(* IEC 61131-3 sources: SmartHomeNew/snapshots/2026-05-19 (part 5) *)

(* ---- PRG_Heating.st ---- *)
PROGRAM PRG_Heating
VAR
    fbHeatingManager : FB_Heating_System_Manager;
    fbDHWManager : FB_DHW_Manager;
    fbDiagnosticsPhase : FB_Heating_Runtime_Diagnostics_Phase;
    fbObserverPhase : FB_Heating_Runtime_Observer_Phase;
    fbMetaSupervisionPublisher : FB_Heating_Runtime_Meta_Supervision_Publisher;
    fbExplainabilityPublisher : FB_Heating_Runtime_Explainability_Publisher;
    fbServiceGatingPhase : FB_Heating_Runtime_Service_Gating_Phase;
    fbStatePublicationPhase : FB_Heating_Runtime_State_Publication_Phase;
    fbOutputProjectionPhase : FB_Heating_Runtime_Output_Projection_Phase;

    L_Runtime_Context : ST_Heating_Runtime_Context;

    L_i : INT;
    L_Current_Hour : UINT;
    L_Boiler_Modulation_REAL : ARRAY[1..GVL_CONSTANTS.C_MAX_BOILERS] OF REAL;
    L_Room_Temps_Normalized : ARRAY[1..GVL_CONSTANTS.C_MAX_ZONES] OF REAL;
    L_Floor_Temps_Normalized : ARRAY[1..GVL_CONSTANTS.C_MAX_HEATING_CIRCUITS] OF REAL;
    L_Outdoor_Temp_Normalized : REAL;

    L_Heating_Emergency_Stop : BOOL;
    L_Heating_Gas_Safety_Stop : BOOL;

    L_Distributed_Execute_Allowed : BOOL;
    L_Distributed_Orchestrate_Allowed : BOOL;
    L_Distributed_Projection_Allowed : BOOL;

    L_Zone_Valves : ARRAY[1..GVL_CONSTANTS.C_MAX_HEATING_CIRCUITS] OF BOOL;
    L_Manifold_Pumps : ARRAY[1..GVL_CONSTANTS.C_MAX_MANIFOLDS] OF BOOL;
    L_Manifold_Valves : ARRAY[1..GVL_CONSTANTS.C_MAX_MANIFOLDS] OF REAL;
    L_Boiler_OT_Enable : ARRAY[1..GVL_CONSTANTS.C_MAX_BOILERS] OF BOOL;
    L_Boiler_OT_Setpoint : ARRAY[1..GVL_CONSTANTS.C_MAX_BOILERS] OF REAL;
    L_Backup_Circulation_Pump : BOOL;
    L_Electric_Heater_Enable : BOOL;
    L_Freeze_Risk_Status : BOOL;
    L_Manifold_Status : ARRAY[1..GVL_CONSTANTS.C_MAX_MANIFOLDS] OF ST_Manifold_Status;
    L_Boiler_Status : ARRAY[1..GVL_CONSTANTS.C_MAX_BOILERS] OF ST_Boiler_Status;
    L_DHW_Heating_Pump : BOOL;
    L_DHW_Circ_Pump : BOOL;
    L_DHW_Status : ST_DHW_Status;
END_VAR

FOR L_i := 1 TO GVL_CONSTANTS.C_MAX_BOILERS DO
    L_Boiler_Modulation_REAL[L_i] := TO_REAL(GVL_IO.AI_Boiler_Modulation[L_i]);
END_FOR;

L_Current_Hour := TO_UINT(GVL_TIME_SERVICE.G_Time_Of_Day_MS / 3600000);

L_Outdoor_Temp_Normalized := GVL_INPUT.IN_Outdoor_Temp;

FOR L_i := 1 TO GVL_CONSTANTS.C_MAX_ZONES DO
    L_Room_Temps_Normalized[L_i] := GVL_INPUT.IN_Room_Temps[L_i];
END_FOR;

FOR L_i := 1 TO GVL_CONSTANTS.C_MAX_HEATING_CIRCUITS DO
    L_Floor_Temps_Normalized[L_i] := GVL_INPUT.IN_Floor_Temps[L_i];
END_FOR;

L_Heating_Emergency_Stop := GVL_COMMAND_SHADOW.G_Heating_Emergency_Stop;
L_Heating_Gas_Safety_Stop := GVL_COMMAND_SHADOW.G_Heating_Gas_Safety_Stop OR GVL_STATE.G_Safety_Gas_Latched;

// Centralized distributed runtime governance.
// Freeze protection and gas safety semantics remain authoritative.
L_Distributed_Execute_Allowed :=
    GVL_Distributed_Execution_Gates.G_Can_Execute;

L_Distributed_Orchestrate_Allowed :=
    GVL_Distributed_Execution_Gates.G_Can_Orchestrate;

L_Distributed_Projection_Allowed :=
    GVL_Distributed_Execution_Gates.G_Can_Own_Projection;

L_Runtime_Context.Runtime_Enabled := TRUE;
L_Runtime_Context.Runtime_Ready := TRUE;
L_Runtime_Context.Runtime_Fault := FALSE;
L_Runtime_Context.Current_Phase := E_Heating_Runtime_Phase.HRP_IDLE;

L_Runtime_Context.Allow_DHW_Phase :=
    L_Distributed_Execute_Allowed;

L_Runtime_Context.Allow_Heating_Phase :=
    L_Distributed_Orchestrate_Allowed;

L_Runtime_Context.Allow_Service_Gating_Phase := TRUE;
L_Runtime_Context.Allow_State_Publication_Phase := TRUE;
L_Runtime_Context.Allow_Diagnostics_Phase := TRUE;

L_Runtime_Context.Allow_Output_Projection_Phase :=
    L_Distributed_Projection_Allowed;

L_Runtime_Context.DHW_Executed := FALSE;
L_Runtime_Context.Heating_Executed := FALSE;
L_Runtime_Context.Service_Gating_Executed := FALSE;
L_Runtime_Context.State_Publication_Executed := FALSE;
L_Runtime_Context.Diagnostics_Executed := FALSE;
L_Runtime_Context.Output_Projection_Executed := FALSE;

L_Runtime_Context.DHW_Before_Heating_Valid := TRUE;
L_Runtime_Context.State_Publication_Before_Diagnostics_Valid := TRUE;
L_Runtime_Context.Output_Projection_Last_Valid := TRUE;

L_Runtime_Context.Diagnostics_Isolation_Valid := TRUE;
L_Runtime_Context.Explainability_Isolation_Valid := TRUE;
L_Runtime_Context.Safety_Isolation_Valid := TRUE;
L_Runtime_Context.OpenTherm_Ownership_Valid := TRUE;
L_Runtime_Context.Cascade_Ownership_Valid := TRUE;

IF NOT L_Distributed_Execute_Allowed THEN
    L_Runtime_Context.Runtime_Status_Code := 20;
    L_Runtime_Context.Runtime_Status_Text :=
        'Heating runtime blocked by distributed governance';
ELSE
    L_Runtime_Context.Runtime_Status_Code := 1;
    L_Runtime_Context.Runtime_Status_Text :=
        'Heating runtime nominal';
END_IF;

L_Runtime_Context.Current_Phase := E_Heating_Runtime_Phase.HRP_IDLE;

fbObserverPhase(
    VI_Authorization_Stage := TRUE,
    VI_Finalization_Stage := FALSE,
    VI_Runtime_Context := L_Runtime_Context,
    VI_Diagnostics_Valid := TRUE
);

IF L_Distributed_Execute_Allowed THEN

    L_Runtime_Context.Current_Phase := E_Heating_Runtime_Phase.HRP_DHW;

    fbDHWManager(
        VI_System_Time_MS := GVL_STATUS.G_System_Time_MS,
        VI_Current_TOD := GVL_STATUS.G_Current_TOD,
        VI_IsActivePLC := GVL_STATUS.G_Is_Active_PLC,
        VI_Temp := GVL_STATE.G_DHW_Temp,
        VI_Pressure := GVL_STATE.G_DHW_Pressure,
        VI_Config := GVL_CONFIG.G_DHW_Config,
        VI_Current_Day_Of_Week := GVL_STATUS.G_Current_Day,
        VI_IO_Modules_Online := GVL_STATUS.G_IO_Modules_Online,
        VI_Reset_Errors := GVL_INTENT_USER.I_Reset_Errors,
        VI_Emergency_Stop := L_Heating_Emergency_Stop,
        VI_System_Mode := GVL_STATE.G_System_Mode,
        VO_Status => L_DHW_Status,
        VO_Heating_Pump => L_DHW_Heating_Pump,
        VO_Circ_Pump => L_DHW_Circ_Pump
    );

    L_Runtime_Context.DHW_Executed := TRUE;

END_IF;

IF L_Heating_Gas_Safety_Stop THEN
    L_DHW_Heating_Pump := FALSE;
    L_DHW_Status.Heating_Pump_On := FALSE;
END_IF;

IF L_Distributed_Orchestrate_Allowed THEN

    L_Runtime_Context.Current_Phase := E_Heating_Runtime_Phase.HRP_HEATING;

    fbHeatingManager(
        VI_System_Mode := GVL_STATE.G_System_Mode,
        VI_System_Time_MS := GVL_STATUS.G_System_Time_MS,
        VI_IsActivePLC := GVL_STATUS.G_Is_Active_PLC,
        VI_Outdoor_Temp := L_Outdoor_Temp_Normalized,
        VI_Config := GVL_CONFIG.G_Heating_Config,
        VI_Tariff := GVL_CONFIG.G_HMI_Tariff_Settings,
        VI_Current_Hour := L_Current_Hour,
        VI_DHW_Heating_Demand := L_DHW_Heating_Pump,
        VI_DHW_Target_Temp := GVL_CONFIG.G_DHW_Config.Target_Temp,
        VI_Emergency_Stop := L_Heating_Emergency_Stop,
        VI_Gas_Safety_Stop := L_Heating_Gas_Safety_Stop,
        VI_Boiler_Error_Status := GVL_STATE.G_Boiler_Error,
        VI_Boiler_OT_Online := GVL_STATE.G_Boiler_OT_Online,
        VI_Boiler_Modulation := L_Boiler_Modulation_REAL,
        VI_Floor_Temps := L_Floor_Temps_Normalized,
        VI_Room_Temps := L_Room_Temps_Normalized,
        VI_Manifold_Pressures := GVL_STATE.G_Manifold_Pressures,
        VI_Manifold_Currents := GVL_STATE.G_Manifold_Currents,
        VI_Manifold_Temps_Supply := GVL_STATE.G_Manifold_T_Supply,
        VI_Manifold_Temps_Return := GVL_STATE.G_Manifold_T_Return,
        VI_Boiler_Flame_Status := GVL_STATE.G_Boiler_Flame,
        VI_Zone_Configs := GVL_CONFIG.G_HMI_FloorHeating_Configs,
        VI_Rule_Actions := GVL_STATE.G_Rule_Actions,
        VI_IO_Modules_Online := GVL_STATUS.G_IO_Modules_Online,
        VI_Manifold_End_Switches := GVL_STATE.G_Manifold_End_Switches,
        VI_Valve_Test_Config := GVL_CONFIG.G_Valve_Test_Config,
        VO_Manifold_Valves => L_Manifold_Valves,
        VO_Manifold_Pumps => L_Manifold_Pumps,
        VO_Zone_Valves => L_Zone_Valves,
        VO_Boiler_OT_Enable => L_Boiler_OT_Enable,
        VO_Boiler_OT_Setpoint => L_Boiler_OT_Setpoint,
        VO_Backup_Circulation_Pump => L_Backup_Circulation_Pump,
        VO_Electric_Heater_Enable => L_Electric_Heater_Enable,
        VO_Freeze_Risk_Status => L_Freeze_Risk_Status,
        VO_Status => L_Manifold_Status,
        VO_Boiler_Status => L_Boiler_Status
    );

    L_Runtime_Context.Heating_Executed := TRUE;

END_IF;

L_Runtime_Context.Current_Phase := E_Heating_Runtime_Phase.HRP_SERVICE_GATING;

fbServiceGatingPhase(
    VI_Enable := TRUE,
    VIO_Manifold_Pumps := L_Manifold_Pumps,
    VIO_Backup_Circulation_Pump := L_Backup_Circulation_Pump,
    VIO_Electric_Heater_Enable := L_Electric_Heater_Enable,
    VIO_DHW_Heating_Pump := L_DHW_Heating_Pump,
    VIO_DHW_Circ_Pump := L_DHW_Circ_Pump,
    VIO_DHW_Status := L_DHW_Status,
    VIO_Freeze_Risk_Status := L_Freeze_Risk_Status
);

L_Runtime_Context.Service_Gating_Executed := fbServiceGatingPhase.VO_Executed;
L_Runtime_Context.Safety_Isolation_Valid := fbServiceGatingPhase.VO_Valid;

L_Runtime_Context.Current_Phase := E_Heating_Runtime_Phase.HRP_STATE_PUBLICATION;

fbStatePublicationPhase(
    VI_Enable := TRUE,
    VI_Zone_Valves := L_Zone_Valves,
    VI_Manifold_Pumps := L_Manifold_Pumps,
    VI_Manifold_Valves := L_Manifold_Valves,
    VI_Boiler_OT_Enable := L_Boiler_OT_Enable,
    VI_Boiler_OT_Setpoint := L_Boiler_OT_Setpoint,
    VI_Backup_Circulation_Pump := L_Backup_Circulation_Pump,
    VI_Electric_Heater_Enable := L_Electric_Heater_Enable,
    VI_Freeze_Risk_Status := L_Freeze_Risk_Status,
    VI_Manifold_Status := L_Manifold_Status,
    VI_Boiler_Status := L_Boiler_Status,
    VI_DHW_Heating_Pump := L_DHW_Heating_Pump,
    VI_DHW_Circ_Pump := L_DHW_Circ_Pump,
    VI_DHW_Status := L_DHW_Status
);

L_Runtime_Context.State_Publication_Executed := fbStatePublicationPhase.VO_Executed;
L_Runtime_Context.State_Publication_Before_Diagnostics_Valid := fbStatePublicationPhase.VO_Valid;

L_Runtime_Context.Current_Phase := E_Heating_Runtime_Phase.HRP_DIAGNOSTICS;

fbDiagnosticsPhase(
    VI_Enable := TRUE,
    VI_System_Time_MS := GVL_STATUS.G_System_Time_MS
);

L_Runtime_Context.Diagnostics_Executed := fbDiagnosticsPhase.VO_Executed;
L_Runtime_Context.Diagnostics_Isolation_Valid := fbDiagnosticsPhase.VO_Valid;

fbObserverPhase(
    VI_Authorization_Stage := FALSE,
    VI_Finalization_Stage := TRUE,
    VI_Runtime_Context := L_Runtime_Context,
    VI_Diagnostics_Valid := L_Runtime_Context.Diagnostics_Isolation_Valid
);

fbMetaSupervisionPublisher(
    VI_Enable := TRUE,
    VI_Runtime_Observation_Valid := GVL_Heating_Runtime_Observation.G_Runtime_Observation_Valid,
    VI_Runtime_Observer_Ready := GVL_Heating_Runtime_Observation.G_Runtime_Observer_Ready,
    VI_Runtime_Observer_Fault := GVL_Heating_Runtime_Observation.G_Runtime_Observer_Fault,
    VI_Runtime_Status_Code := GVL_Heating_Runtime_Observation.G_Runtime_Observation_Status_Code,
    VI_Runtime_Status_Text := GVL_Heating_Runtime_Observation.G_Runtime_Observation_Status_Text
);

GVL_Heating_Runtime_Meta.G_Runtime_Meta_Supervision :=
    fbMetaSupervisionPublisher.VO_Meta;

GVL_Heating_Runtime_Meta.G_Runtime_Meta_Publication_Valid :=
    fbMetaSupervisionPublisher.VO_Publication_Valid;

GVL_Heating_Runtime_Meta.G_Runtime_Meta_Status_Code :=
    fbMetaSupervisionPublisher.VO_Meta.Status_Code;

GVL_Heating_Runtime_Meta.G_Runtime_Meta_Status_Text :=
    fbMetaSupervisionPublisher.VO_Meta.Status_Text;

fbExplainabilityPublisher(
    VI_Enable := TRUE,
    VI_System_Time_MS := GVL_STATUS.G_System_Time_MS,
    VI_Runtime_Context := L_Runtime_Context,
    VI_Runtime_Observation_Valid := GVL_Heating_Runtime_Observation.G_Runtime_Observation_Valid,
    VI_Runtime_Observer_Fault := GVL_Heating_Runtime_Observation.G_Runtime_Observer_Fault,
    VI_Runtime_Status_Code := GVL_Heating_Runtime_Observation.G_Runtime_Observation_Status_Code,
    VI_Runtime_Status_Text := GVL_Heating_Runtime_Observation.G_Runtime_Observation_Status_Text
);

GVL_Heating_Runtime_Explainability.G_Runtime_Phase_Event :=
    fbExplainabilityPublisher.VO_Phase_Event;

GVL_Heating_Runtime_Explainability.G_Runtime_Anomaly :=
    fbExplainabilityPublisher.VO_Anomaly;

GVL_Heating_Runtime_Explainability.G_Runtime_Blackbox_Event :=
    fbExplainabilityPublisher.VO_Blackbox_Event;

GVL_Heating_Runtime_Explainability.G_Runtime_Blackbox_Timeline :=
    fbExplainabilityPublisher.VO_Blackbox_Timeline;

GVL_Heating_Runtime_Explainability.G_Runtime_Event_Buffer :=
    fbExplainabilityPublisher.VO_Event_Buffer;

GVL_Heating_Runtime_Explainability.G_Runtime_Adaptive_Intelligence :=
    fbExplainabilityPublisher.VO_Adaptive_Intelligence;

GVL_Heating_Runtime_Explainability.G_Runtime_Causality_Graph :=
    fbExplainabilityPublisher.VO_Causality_Graph;

GVL_Heating_Runtime_Explainability.G_Runtime_Explainability_Publication_Valid :=
    fbExplainabilityPublisher.VO_Publication_Valid;

GVL_Heating_Runtime_Explainability.G_Runtime_Explainability_Status_Code :=
    fbExplainabilityPublisher.VO_Phase_Event.Status_Code;

GVL_Heating_Runtime_Explainability.G_Runtime_Explainability_Status_Text :=
    fbExplainabilityPublisher.VO_Phase_Event.Status_Text;

IF L_Distributed_Projection_Allowed THEN

    L_Runtime_Context.Current_Phase := E_Heating_Runtime_Phase.HRP_OUTPUT_PROJECTION;

    fbOutputProjectionPhase(
        VI_Enable := TRUE,
        VI_Zone_Valves := L_Zone_Valves,
        VI_Manifold_Pumps := L_Manifold_Pumps,
        VI_Manifold_Valves := L_Manifold_Valves,
        VI_DHW_Heating_Pump := L_DHW_Heating_Pump,
        VI_DHW_Circ_Pump := L_DHW_Circ_Pump,
        VI_Backup_Circulation_Pump := L_Backup_Circulation_Pump,
        VI_Electric_Heater_Enable := L_Electric_Heater_Enable
    );

    L_Runtime_Context.Output_Projection_Executed :=
        fbOutputProjectionPhase.VO_Executed;

    L_Runtime_Context.Output_Projection_Last_Valid :=
        fbOutputProjectionPhase.VO_Valid;

END_IF;

L_Runtime_Context.Current_Phase := E_Heating_Runtime_Phase.HRP_COMPLETE;

// >>> BULK_SYNC_ANCHOR: PRG_Heating <<<
END_PROGRAM

(* ---- PRG_Heating_Policy_Manager.st ---- *)
PROGRAM PRG_Heating_Policy_Manager
VAR
    fbPolicyManager : FB_Heating_Policy_Manager;
    fbSchedule : FB_Heating_Schedule_Preheat;
    fbThermal : FB_Heating_Thermal_Model;
    fbPredictive : FB_Heating_Predictive_Controller;
    fbOptimizer : FB_Heating_Optimizer;
    fbTime : FB_Time_Service;
    L_i : INT;
    L_Room_Avg : REAL;
    L_Floor_Avg : REAL;
END_VAR

fbTime();
fbThermal();
fbPredictive();
fbOptimizer();

L_Room_Avg := 0.0;
L_Floor_Avg := 0.0;

FOR L_i := 1 TO GVL_CONSTANTS.C_MAX_ZONES DO
    L_Room_Avg := L_Room_Avg + GVL_STATE.G_Room_Temps[L_i];
    L_Floor_Avg := L_Floor_Avg + GVL_STATE.G_Floor_Temps[L_i];
END_FOR;

L_Room_Avg := L_Room_Avg / TO_REAL(GVL_CONSTANTS.C_MAX_ZONES);
L_Floor_Avg := L_Floor_Avg / TO_REAL(GVL_CONSTANTS.C_MAX_ZONES);

fbPolicyManager(
    VI_System_Time_MS := GVL_TIME_SERVICE.G_Now_MS,
    VI_System_Mode := GVL_STATE.G_System_Mode,
    VI_RootCause := GVL_STATE.G_Heating_RootCause,
    VI_RootConfidence := GVL_STATE.G_Heating_RootConfidence,
    VI_Min_Hold_MS := GVL_CONFIG.G_Policy_Min_Hold_MS,
    VI_Emergency_Stop := GVL_STATE.G_Safety_Emergency_Stop,
    VI_Gas_Safety := GVL_STATE.G_Safety_Gas_Latched,
    VI_Room_Temp_Avg := L_Room_Avg,
    VI_Floor_Temp_Avg := L_Floor_Avg,
    VI_Supply_Temp := GVL_STATE.G_Manifold_T_Supply[1],
    VI_Return_Temp := GVL_STATE.G_Manifold_T_Return[1],
    VI_Target_Temp := GVL_STATE.G_Target_Temperature,
    VI_Room_Temps := GVL_STATE.G_Room_Temps,
    VI_Floor_Temps := GVL_STATE.G_Floor_Temps
);

fbSchedule(
    VI_System_Time_MS := GVL_TIME_SERVICE.G_Now_MS,
    VI_Time_Of_Day_MS := GVL_TIME_SERVICE.G_Time_Of_Day_MS,
    VI_Day_Of_Week := GVL_TIME_SERVICE.G_Day_Of_Week,
    VI_Enable := TRUE
);

GVL_HEATING_POLICY.G_Policy_Mode := fbPolicyManager.VO_Policy_Mode;
GVL_HEATING_POLICY.G_Policy_Block_Heating_Request := fbPolicyManager.VO_Block_Heating;
GVL_HEATING_POLICY.G_Policy_Target_Adjustment := fbPolicyManager.VO_Target_Adjustment;
GVL_HEATING_POLICY.G_Policy_Priority_Multiplier := fbPolicyManager.VO_Priority_Multiplier;
GVL_HEATING_POLICY.G_Policy_Self_Tune_Active := fbPolicyManager.VO_Self_Tune_Active;
GVL_HEATING_POLICY.G_Policy_Self_Tune_Level := fbPolicyManager.VO_Self_Tune_Level;
GVL_HEATING_POLICY.G_Policy_Feedback_Stable := fbPolicyManager.VO_Feedback_Stable;
GVL_HEATING_POLICY.G_Policy_Feedback_Improving := fbPolicyManager.VO_Feedback_Improving;
GVL_HEATING_POLICY.G_Policy_Feedback_Quality := fbPolicyManager.VO_Feedback_Quality;

END_PROGRAM

(* ---- PRG_Historical_Ordering_Integrity_Governor.st ---- *)
PROGRAM PRG_Historical_Ordering_Integrity_Governor
IF GVL_DISTRIBUTED_EPOCH_LINEARITY_FABRIC.Distributed_Epoch_Linearity_Granted
AND NOT GVL_HISTORICAL_ORDERING_INTEGRITY_FABRIC.Historical_Order_Divergence
AND NOT GVL_HISTORICAL_ORDERING_INTEGRITY_FABRIC.Unsafe_Historical_Rewrite_Detected
AND NOT GVL_HISTORICAL_ORDERING_INTEGRITY_FABRIC.Historical_Causality_Gap_Detected THEN

    GVL_HISTORICAL_ORDERING_INTEGRITY_FABRIC.Historical_Ordering_Integrity_Valid := TRUE;
    GVL_HISTORICAL_ORDERING_INTEGRITY_FABRIC.Historical_Ordering_Integrity_Granted := TRUE;
    GVL_HISTORICAL_ORDERING_INTEGRITY_FABRIC.Historical_Ordering_Integrity_Granted_Proof := TRUE;
    GVL_HISTORICAL_ORDERING_INTEGRITY_FABRIC.Historical_Timeline_Canonical := TRUE;
    GVL_HISTORICAL_ORDERING_INTEGRITY_FABRIC.Forensic_Ordering_Coherent := TRUE;
END_IF;
END_PROGRAM

(* ---- PRG_IO_Write.st ---- *)
PROGRAM PRG_IO_Write
VAR
    L_i : INT;
    L_Heating_Forced_Off : BOOL;
    L_Vent_Forced_Off : BOOL;
    L_Water_Forced_Off : BOOL;
    L_Access_Forced_Off : BOOL;
    L_Access_Safety_Override : BOOL;
    L_Global_Hard_Stop : BOOL;
    L_Gas_Safety_Stop : BOOL;
    L_Freeze_Active : BOOL;
    L_Gas_Fire_Siren_Enable : BOOL;
    L_PreOutput_Block_IO : BOOL;
    L_Output_Freshness_Block : BOOL;
    L_Output_Publication_Block : BOOL;
    L_Distributed_Publication_Block : BOOL;
    L_Snapshot_Block : BOOL;
    L_Distributed_Execution_Block : BOOL;
    L_Gas_Siren_Authority : BOOL;
    L_Fire_Siren_Authority : BOOL;
    fbTrace : FB_Trace_Write;
END_VAR

L_PreOutput_Block_IO := GVL_COMMAND_VERIFY.PreOutput_Block_IO;
L_Output_Freshness_Block := GVL_OUTPUT_EPOCH.Output_Forced_Safe_Decay;

L_Output_Publication_Block :=
    (NOT GVL_OUTPUT_EPOCH.Output_Publication_Valid)
    OR (NOT GVL_OUTPUT_EPOCH.Output_Runtime_Epoch_Valid)
    OR GVL_OUTPUT_EPOCH.Output_Lease_Expired;

// Final distributed publication continuity authority.
L_Distributed_Publication_Block :=
    (NOT GVL_DISTRIBUTED_COMMIT.Distributed_Commit_Valid)
    OR GVL_DISTRIBUTED_COMMIT.Distributed_Commit_Quarantine_Active
    OR GVL_DISTRIBUTED_COMMIT.Commit_Lease_Expired
    OR (NOT GVL_DISTRIBUTED_SNAPSHOT.Distributed_Publication_Reconciled)
    OR (NOT GVL_DISTRIBUTED_SNAPSHOT.Distributed_Publication_Freeze_Valid)
    OR (NOT GVL_DISTRIBUTED_SNAPSHOT.Distributed_Snapshot_Consistent);

L_Snapshot_Block :=
    (NOT GVL_RUNTIME_SNAPSHOT.Snapshot_Frozen)
    OR (NOT GVL_RUNTIME_SNAPSHOT.Snapshot_Publication_Allowed)
    OR (NOT GVL_RUNTIME_SNAPSHOT.Snapshot_Copy_Valid)
    OR (NOT GVL_RUNTIME_SNAPSHOT.Snapshot_Isolation_Valid)
    OR GVL_RUNTIME_SNAPSHOT.Snapshot_Mutation_Detected;

L_Distributed_Execution_Block :=
    NOT GVL_Distributed_Execution_Gates.G_Can_Execute
    OR NOT GVL_Distributed_Execution_Gates.G_Can_Own_Projection;

L_Global_Hard_Stop :=
    GVL_COMMAND_SHADOW.G_Heating_Emergency_Stop
    OR L_PreOutput_Block_IO
    OR L_Output_Freshness_Block
    OR L_Output_Publication_Block
    OR L_Distributed_Publication_Block
    OR L_Snapshot_Block
    OR L_Distributed_Execution_Block;

L_Gas_Safety_Stop := GVL_COMMAND_SHADOW.G_Heating_Gas_Safety_Stop OR GVL_COMMAND_SHADOW.G_Boiler_Stop;
L_Freeze_Active := GVL_STATE.G_Safety_Freeze_Risk;
L_Gas_Fire_Siren_Enable := GVL_ALARM.G_Gas_Fire_Siren OR GVL_ALARM.G_Global_Siren OR GVL_ALARM.G_Global_Critical;

L_Gas_Siren_Authority := GVL_HEALTH_BRIDGE.G_Gas_Detected OR GVL_HEALTH_BRIDGE.G_CO_Alarm_Level OR GVL_STATE.G_Safety_Gas_Latched;
L_Fire_Siren_Authority := GVL_HEALTH_BRIDGE.G_Smoke_Detected OR GVL_STATE.G_Safety_Smoke_Latched;

IF NOT GVL_STATUS.G_Is_Active_PLC OR L_Global_Hard_Stop THEN

    FOR L_i := 1 TO GVL_CONSTANTS.C_MAX_HEATING_CIRCUITS DO
        GVL_IO.DO_Zone_Valves[L_i] := FALSE;
    END_FOR;

    GVL_IO.DO_Gas_Valve_Close := TRUE;

    IF L_Distributed_Publication_Block THEN
        fbTrace(
            iLayer := TRACE_IO,
            iSource := SRC_IO,
            iReason := REASON_SAFETY_BLOCK,
            iValueBool := TRUE,
            iValueReal := UDINT_TO_REAL(GVL_DISTRIBUTED_COMMIT.Distributed_Commit_Last_Error_Code),
            iText := 'IO blocked by distributed publication continuity authority');
    END_IF;

    IF L_Output_Publication_Block THEN
        fbTrace(
            iLayer := TRACE_IO,
            iSource := SRC_IO,
            iReason := REASON_SAFETY_BLOCK,
            iValueBool := TRUE,
            iValueReal := UDINT_TO_REAL(GVL_OUTPUT_EPOCH.Output_Last_Error_Code),
            iText := 'IO blocked by finalized output publication authority');
    END_IF;

    RETURN;
END_IF;

fbTrace(
    iLayer := TRACE_IO,
    iSource := SRC_IO,
    iReason := REASON_DOMAIN_PROJECTION,
    iValueBool := TRUE,
    iValueReal := 0.0,
    iText := 'IO write projection executed');
END_PROGRAM

(* ---- PRG_Meta_Governance_Governor.st ---- *)
PROGRAM PRG_Meta_Governance_Governor
VAR
    L_Now_MS : UDINT;
    L_Meta_Valid : BOOL := TRUE;
    L_Error_Code : UDINT := 0;
    L_Error_Text : STRING(160) := '';
END_VAR

L_Now_MS := GVL_STATUS.G_System_Time_MS;
L_Meta_Valid := TRUE;
L_Error_Code := 0;
L_Error_Text := '';

// Fail-safe defaults.
GVL_META_GOVERNANCE_FABRIC.Meta_Governance_Valid := FALSE;
GVL_META_GOVERNANCE_FABRIC.Meta_Governance_Granted := FALSE;
GVL_META_GOVERNANCE_FABRIC.Meta_Governance_Quarantine_Active := TRUE;

GVL_META_GOVERNANCE_FABRIC.Governance_Graph_Acyclic := FALSE;
GVL_META_GOVERNANCE_FABRIC.Authority_Rooting_Valid := FALSE;
GVL_META_GOVERNANCE_FABRIC.Independent_Validation_Preserved := FALSE;
GVL_META_GOVERNANCE_FABRIC.Meta_Consistency_Coherent := FALSE;
GVL_META_GOVERNANCE_FABRIC.Recursive_Trust_Boundaries_Stable := FALSE;

// Epistemic integrity required.
IF NOT GVL_EPISTEMIC_INTEGRITY_FABRIC.Epistemic_Integrity_Granted THEN
    L_Meta_Valid := FALSE;
    L_Error_Code := 45000;
    L_Error_Text := 'Epistemic integrity authority not granted';
END_IF;

// Meta-governance recursion detectors.
IF GVL_META_GOVERNANCE_FABRIC.Recursive_Authority_Dependency_Detected THEN
    L_Meta_Valid := FALSE;
    L_Error_Code := 45001;
    L_Error_Text := 'Recursive authority dependency detected';
END_IF;

IF GVL_META_GOVERNANCE_FABRIC.Circular_Validation_Chain_Detected THEN
    L_Meta_Valid := FALSE;
    L_Error_Code := 45002;
    L_Error_Text := 'Circular validation chain detected';
END_IF;

IF GVL_META_GOVERNANCE_FABRIC.SelfJustifying_Governance_State_Detected THEN
    L_Meta_Valid := FALSE;
    L_Error_Code := 45003;
    L_Error_Text := 'Self-justifying governance state detected';
END_IF;

IF GVL_META_GOVERNANCE_FABRIC.Epistemic_Recursion_Leakage_Detected THEN
    L_Meta_Valid := FALSE;
    L_Error_Code := 45004;
    L_Error_Text := 'Epistemic recursion leakage detected';
END_IF;

IF GVL_META_GOVERNANCE_FABRIC.Authority_Bootstrap_Paradox_Detected THEN
    L_Meta_Valid := FALSE;
    L_Error_Code := 45005;
    L_Error_Text := 'Authority bootstrap paradox detected';
END_IF;

IF GVL_META_GOVERNANCE_FABRIC.Meta_Consistency_Erosion_Detected THEN
    L_Meta_Valid := FALSE;
    L_Error_Code := 45006;
    L_Error_Text := 'Meta-consistency erosion detected';
END_IF;

// Meta-governance consistency validation.
IF L_Meta_Valid
AND NOT GVL_META_GOVERNANCE_FABRIC.Validator_Independence_Valid THEN
    L_Meta_Valid := FALSE;
    L_Error_Code := 45010;
    L_Error_Text := 'Validator independence invalid';
END_IF;

IF L_Meta_Valid
AND NOT GVL_META_GOVERNANCE_FABRIC.CrossLayer_Causality_Grounded THEN
    L_Meta_Valid := FALSE;
    L_Error_Code := 45011;
    L_Error_Text := 'Cross-layer causality grounding invalid';
END_IF;

IF L_Meta_Valid
AND NOT GVL_META_GOVERNANCE_FABRIC.Bootstrap_Validation_Absent THEN
    L_Meta_Valid := FALSE;
    L_Error_Code := 45012;
    L_Error_Text := 'Bootstrap validation absence invalid';
END_IF;

IF L_Meta_Valid
AND NOT GVL_META_GOVERNANCE_FABRIC.SelfReference_Elimination_Valid THEN
    L_Meta_Valid := FALSE;
    L_Error_Code := 45013;
    L_Error_Text := 'Self-reference elimination invalid';
END_IF;

IF L_Meta_Valid THEN
    GVL_META_GOVERNANCE_FABRIC.Meta_Governance_Valid := TRUE;
    GVL_META_GOVERNANCE_FABRIC.Meta_Governance_Granted := TRUE;
    GVL_META_GOVERNANCE_FABRIC.Meta_Governance_Quarantine_Active := FALSE;

    GVL_META_GOVERNANCE_FABRIC.Governance_Graph_Acyclic := TRUE;
    GVL_META_GOVERNANCE_FABRIC.Authority_Rooting_Valid := TRUE;
    GVL_META_GOVERNANCE_FABRIC.Independent_Validation_Preserved := TRUE;
    GVL_META_GOVERNANCE_FABRIC.Meta_Consistency_Coherent := TRUE;
    GVL_META_GOVERNANCE_FABRIC.Recursive_Trust_Boundaries_Stable := TRUE;

    GVL_META_GOVERNANCE_FABRIC.Meta_Governance_Epoch :=
        GVL_EPISTEMIC_INTEGRITY_FABRIC.Epistemic_Integrity_Epoch;

    GVL_META_GOVERNANCE_FABRIC.Meta_Governance_Epoch_Coherent := TRUE;

    GVL_META_GOVERNANCE_FABRIC.Meta_Governance_Last_Update_MS :=
        L_Now_MS;

    GVL_META_GOVERNANCE_FABRIC.Meta_Governance_Lease_Expired := FALSE;

    GVL_META_GOVERNANCE_FABRIC.Meta_Governance_Last_Error_Code := 0;
    GVL_META_GOVERNANCE_FABRIC.Meta_Governance_Last_Error_Text := '';
ELSE
    GVL_META_GOVERNANCE_FABRIC.Meta_Governance_Valid := FALSE;
    GVL_META_GOVERNANCE_FABRIC.Meta_Governance_Granted := FALSE;
    GVL_META_GOVERNANCE_FABRIC.Meta_Governance_Quarantine_Active := TRUE;

    GVL_META_GOVERNANCE_FABRIC.Meta_Governance_Lease_Expired := TRUE;

    GVL_META_GOVERNANCE_FABRIC.Meta_Governance_Last_Error_Code :=
        L_Error_Code;

    GVL_META_GOVERNANCE_FABRIC.Meta_Governance_Last_Error_Text :=
        L_Error_Text;

    GVL_META_GOVERNANCE_FABRIC.Meta_Governance_Invalidation_Count :=
        GVL_META_GOVERNANCE_FABRIC.Meta_Governance_Invalidation_Count + 1;
END_IF;

END_PROGRAM

(* ---- PRG_Mode_Manager.st ---- *)
PROGRAM PRG_Mode_Manager
VAR
    fbMode : FB_Mode_Manager;
    L_Last_Mode : E_Behavior_Mode := BEHAVIOR_HOME;
END_VAR

fbMode(
    VI_Is_Night := GVL_STATUS.G_Is_Night,
    VI_Away_Request := GVL_MODE.G_Away_Request OR GVL_PRESENCE.G_Auto_Away_Request,
    VI_Maintenance_Request := GVL_MODE.G_Maintenance_Request,
    VI_System_Time_MS := GVL_STATUS.G_System_Time_MS
);

GVL_MODE.G_Current_Behavior_Mode := fbMode.VO_Mode;
GVL_MODE.G_Mode_Code := fbMode.VO_Mode_Code;

IF L_Last_Mode <> fbMode.VO_Mode THEN
    GVL_MODE.G_Mode_Last_Change_TS := GVL_STATUS.G_System_Time_MS;
    L_Last_Mode := fbMode.VO_Mode;
END_IF;
END_PROGRAM

(* ---- PRG_OpenTherm_Adapter_Status.st ---- *)
PROGRAM PRG_OpenTherm_Adapter_Status
VAR
    L_i : INT;
    L_Now_MS : UDINT;
    L_Heartbeat_Age : UDINT;
    L_Command_Age : UDINT;
END_VAR

L_Now_MS := GVL_STATUS.G_System_Time_MS;

FOR L_i := 1 TO GVL_CONSTANTS.C_MAX_BOILERS DO

    // ======================================================
    // HEARTBEAT VALIDATION
    // ======================================================
    IF GVL_OPENTHERM_ADAPTER.G_Status[L_i].Raw_Heartbeat <>
       GVL_OPENTHERM_ADAPTER.G_Status[L_i].Last_Heartbeat THEN

        GVL_OPENTHERM_ADAPTER.G_Status[L_i].Last_Heartbeat :=
            GVL_OPENTHERM_ADAPTER.G_Status[L_i].Raw_Heartbeat;

        GVL_OPENTHERM_ADAPTER.G_Status[L_i].Last_Heartbeat_MS := L_Now_MS;
    END_IF;

    L_Heartbeat_Age :=
        L_Now_MS - GVL_OPENTHERM_ADAPTER.G_Status[L_i].Last_Heartbeat_MS;

    GVL_OPENTHERM_ADAPTER.G_Status[L_i].Heartbeat_Age_MS :=
        L_Heartbeat_Age;

    GVL_OPENTHERM_ADAPTER.G_Status[L_i].Heartbeat_Timeout :=
        (L_Heartbeat_Age > GVL_CONFIG.G_OpenTherm_Heartbeat_Timeout_MS);

    // ======================================================
    // COMMAND ACK VALIDATION
    // ======================================================
    GVL_OPENTHERM_ADAPTER.G_Status[L_i].Command_Ack :=
        (GVL_OPENTHERM_ADAPTER.G_Status[L_i].Raw_Ack_Seq =
         GVL_OPENTHERM_ADAPTER.G_Command[L_i].Sequence);

    GVL_OPENTHERM_ADAPTER.G_Status[L_i].Last_Command_Ack_Seq :=
        GVL_OPENTHERM_ADAPTER.G_Status[L_i].Raw_Ack_Seq;

    L_Command_Age :=
        L_Now_MS - GVL_OPENTHERM_ADAPTER.G_Command[L_i].Last_Write_MS;

    GVL_OPENTHERM_ADAPTER.G_Status[L_i].Command_Age_MS :=
        L_Command_Age;

    GVL_OPENTHERM_ADAPTER.G_Status[L_i].Command_Timeout :=
        (NOT GVL_OPENTHERM_ADAPTER.G_Status[L_i].Command_Ack) AND
        (L_Command_Age > GVL_CONFIG.G_OpenTherm_Command_Ack_Timeout_MS);

    // ======================================================
    // FINAL ADAPTER STATE
    // ======================================================
    GVL_OPENTHERM_ADAPTER.G_Status[L_i].Adapter_Online :=
        GVL_OPENTHERM_ADAPTER.G_Status[L_i].Raw_Online AND
        (NOT GVL_OPENTHERM_ADAPTER.G_Status[L_i].Heartbeat_Timeout) AND
        (NOT GVL_OPENTHERM_ADAPTER.G_Status[L_i].Command_Timeout);

    GVL_OPENTHERM_ADAPTER.G_Status[L_i].Adapter_Error :=
        GVL_OPENTHERM_ADAPTER.G_Status[L_i].Raw_Error OR
        GVL_OPENTHERM_ADAPTER.G_Status[L_i].Command_Timeout OR
        GVL_OPENTHERM_ADAPTER.G_Status[L_i].Heartbeat_Timeout;

    // ======================================================
    // ENUM STATES
    // ======================================================
    IF GVL_OPENTHERM_ADAPTER.G_Status[L_i].Heartbeat_Timeout THEN
        GVL_OPENTHERM_ADAPTER.G_Status[L_i].Adapter_State := OT_STATE_HEARTBEAT_TIMEOUT;
        GVL_OPENTHERM_ADAPTER.G_Status[L_i].Error_State := OT_ERROR_HEARTBEAT_TIMEOUT;

    ELSIF GVL_OPENTHERM_ADAPTER.G_Status[L_i].Command_Timeout THEN
        GVL_OPENTHERM_ADAPTER.G_Status[L_i].Adapter_State := OT_STATE_ACK_TIMEOUT;
        GVL_OPENTHERM_ADAPTER.G_Status[L_i].Error_State := OT_ERROR_ACK_TIMEOUT;

    ELSIF GVL_OPENTHERM_ADAPTER.G_Status[L_i].Raw_Error THEN
        GVL_OPENTHERM_ADAPTER.G_Status[L_i].Adapter_State := OT_STATE_ADAPTER_ERROR;
        GVL_OPENTHERM_ADAPTER.G_Status[L_i].Error_State := OT_ERROR_ADAPTER_FAULT;

    ELSIF GVL_OPENTHERM_ADAPTER.G_Status[L_i].Adapter_Online THEN
        GVL_OPENTHERM_ADAPTER.G_Status[L_i].Adapter_State := OT_STATE_ONLINE;
        GVL_OPENTHERM_ADAPTER.G_Status[L_i].Error_State := OT_ERROR_NONE;

    ELSE
        GVL_OPENTHERM_ADAPTER.G_Status[L_i].Adapter_State := OT_STATE_OFFLINE;
        GVL_OPENTHERM_ADAPTER.G_Status[L_i].Error_State := OT_ERROR_COMMUNICATION;
    END_IF;

    // ======================================================
    // PUBLISH TO SYSTEM STATE
    // ======================================================
    GVL_STATE.G_Boiler_OT_Online[L_i] :=
        GVL_OPENTHERM_ADAPTER.G_Status[L_i].Adapter_Online;

    GVL_STATE.G_Boiler_OT_Command_Ack[L_i] :=
        GVL_OPENTHERM_ADAPTER.G_Status[L_i].Command_Ack;

    GVL_STATE.G_Boiler_OT_Command_Timeout[L_i] :=
        GVL_OPENTHERM_ADAPTER.G_Status[L_i].Command_Timeout;

    GVL_STATE.G_Boiler_OT_Heartbeat_Timeout[L_i] :=
        GVL_OPENTHERM_ADAPTER.G_Status[L_i].Heartbeat_Timeout;

    GVL_STATE.G_Boiler_OT_Adapter_Error[L_i] :=
        GVL_OPENTHERM_ADAPTER.G_Status[L_i].Adapter_Error;

    GVL_STATE.G_Boiler_OT_Heartbeat_Age_MS[L_i] :=
        GVL_OPENTHERM_ADAPTER.G_Status[L_i].Heartbeat_Age_MS;

    GVL_STATE.G_Boiler_OT_Command_Age_MS[L_i] :=
        GVL_OPENTHERM_ADAPTER.G_Status[L_i].Command_Age_MS;

    GVL_STATE.G_Boiler_OT_Adapter_State[L_i] :=
        GVL_OPENTHERM_ADAPTER.G_Status[L_i].Adapter_State;

    GVL_STATE.G_Boiler_OT_Error_State[L_i] :=
        GVL_OPENTHERM_ADAPTER.G_Status[L_i].Error_State;

    GVL_STATE.G_Boiler_Error[L_i] :=
        GVL_OPENTHERM_ADAPTER.G_Status[L_i].Adapter_Error;

    GVL_STATE.G_Boiler_Flame[L_i] :=
        GVL_OPENTHERM_ADAPTER.G_Status[L_i].Raw_Flame;

END_FOR;

END_PROGRAM

(* ---- PRG_Passive_Runtime_Verification_Governor.st ---- *)
PROGRAM PRG_Passive_Runtime_Verification_Governor
// PASSIVE READ-ONLY OBSERVABILITY GOVERNOR
// NO authority mutation
// NO execution mutation
// NO blocking semantics

GVL_PASSIVE_RUNTIME_VERIFICATION_FABRIC.Runtime_Verification_Consistency_Valid :=
    GVL_CAUSALITY_REVERSAL_PREVENTION_FABRIC.Causality_Reversal_Prevention_Granted;

GVL_PASSIVE_RUNTIME_VERIFICATION_FABRIC.Runtime_Verification_Lineage_Coherent := TRUE;
GVL_PASSIVE_RUNTIME_VERIFICATION_FABRIC.Runtime_Verification_Timeline_Monotonic := TRUE;

END_PROGRAM

(* ---- PRG_Peer_Heartbeat_Ingestion.st ---- *)
PROGRAM PRG_Peer_Heartbeat_Ingestion
VAR
    L_Now_MS : UDINT;
END_VAR

// ======================================================
// PEER HEARTBEAT INGESTION
// ======================================================
// Bounded transport/heartbeat ingestion bridge.
//
// Purpose:
// map physical partner heartbeat inputs into runtime-visible
// remote PLC liveness state consumed by arbitration layers.
//
// This layer does NOT:
// - perform distributed epoch reconciliation
// - publish peer fencing tokens
// - mutate distributed authority state
// - participate in runtime/output hard-stop governance
//
// Ownership:
// physical partner inputs  -> GVL_IO
// heartbeat ingestion      -> this PRG
// arbitration/governance   -> downstream consumers only
// ======================================================

L_Now_MS := GVL_STATUS.G_System_Time_MS;

// ------------------------------------------------------
// Physical heartbeat ingestion.
// ------------------------------------------------------

GVL_STATUS.G_Remote_PLC_Pulse := GVL_IO.DI_Partner_Pulse;

// ------------------------------------------------------
// Partner active visibility projection.
// ------------------------------------------------------

IF GVL_IO.DI_Partner_Active THEN
    GVL_STATUS.G_Remote_PLC_Last_Seen_MS := L_Now_MS;
END_IF;

// ------------------------------------------------------
// Optional pulse freshness refresh.
// ------------------------------------------------------

IF GVL_IO.DI_Partner_Pulse THEN
    GVL_STATUS.G_Remote_PLC_Last_Seen_MS := L_Now_MS;
END_IF;

// ------------------------------------------------------
// Remote liveness projection.
// ------------------------------------------------------

GVL_STATUS.G_Remote_PLC_Alive :=
    (L_Now_MS - GVL_STATUS.G_Remote_PLC_Last_Seen_MS) < 3000;

// >>> BULK_SYNC_ANCHOR: PRG_Peer_Heartbeat_Ingestion <<<
END_PROGRAM

(* ---- PRG_Peer_Session_Publication.st ---- *)
PROGRAM PRG_Peer_Session_Publication
// ======================================================
// PEER SESSION PUBLICATION
// ======================================================
// Canonical local PLC session export.
//
// Purpose:
// publish normalized runtime/session authority state into
// explicit peer-session transport contract surface.
//
// This layer does NOT:
// - perform network replication
// - perform distributed reconciliation
// - consume remote peer state
//
// Future transport/replication layers may replicate these
// fields to partner PLCs or external HA channels.
// ======================================================

GVL_PEER_SESSION.Remote_Session_Valid :=
    GVL_RUNTIME_EPOCH.Runtime_Runtime_Barrier_OK
    AND GVL_RUNTIME_EPOCH.Runtime_IO_Publication_Allowed;

GVL_PEER_SESSION.Remote_Last_Refresh_MS :=
    GVL_STATUS.G_System_Time_MS;

GVL_PEER_SESSION.Remote_Runtime_Epoch :=
    GVL_RUNTIME_EPOCH.Runtime_Epoch;

GVL_PEER_SESSION.Remote_Snapshot_Epoch :=
    GVL_RUNTIME_SNAPSHOT.Snapshot_Epoch;

GVL_PEER_SESSION.Remote_Boot_Generation :=
    GVL_TIME_MONOTONIC.Boot_Generation_ID;

GVL_PEER_SESSION.Remote_Fencing_Token :=
    GVL_PLC_FENCING.PLC_Fencing_Token;

GVL_PEER_SESSION.Remote_Publication_Allowed :=
    GVL_OUTPUT_EPOCH.Output_Publication_Valid
    AND NOT GVL_OUTPUT_EPOCH.Output_Forced_Safe_Decay;

GVL_PEER_SESSION.Remote_Runtime_Healthy :=
    GVL_RUNTIME_EPOCH.Runtime_Runtime_Barrier_OK;

// >>> BULK_SYNC_ANCHOR: PRG_Peer_Session_Publication <<<
END_PROGRAM

(* ---- PRG_Physical_Transaction_Governor.st ---- *)
PROGRAM PRG_Physical_Transaction_Governor
VAR
    L_Now_MS : UDINT;
    L_Transaction_Valid : BOOL := TRUE;
    L_Error_Code : UDINT := 0;
    L_Error_Text : STRING(160) := '';
END_VAR

L_Now_MS := GVL_STATUS.G_System_Time_MS;
L_Transaction_Valid := TRUE;
L_Error_Code := 0;
L_Error_Text := '';

// Fail-safe defaults.
GVL_PHYSICAL_TRANSACTION.Physical_Transaction_Valid := FALSE;
GVL_PHYSICAL_TRANSACTION.Physical_Transaction_Granted := FALSE;
GVL_PHYSICAL_TRANSACTION.Physical_Transaction_Quarantine_Active := TRUE;

GVL_PHYSICAL_TRANSACTION.All_Actuators_Converged := FALSE;
GVL_PHYSICAL_TRANSACTION.Cross_Actuator_Epoch_Coherent := FALSE;
GVL_PHYSICAL_TRANSACTION.Distributed_Actuation_Coherent := FALSE;
GVL_PHYSICAL_TRANSACTION.Stable_Plant_State_Confirmed := FALSE;

// Bind transaction epochs.
GVL_PHYSICAL_TRANSACTION.Physical_Transaction_Command_Epoch :=
    GVL_ACTUATION_AUTHORITY.Actuation_Command_Epoch;

GVL_PHYSICAL_TRANSACTION.Physical_Transaction_ACK_Epoch :=
    GVL_ACTUATION_AUTHORITY.Field_ACK_Epoch;

IF GVL_PHYSICAL_TRANSACTION.Physical_Transaction_Command_Epoch <>
   GVL_PHYSICAL_TRANSACTION.Physical_Transaction_ACK_Epoch THEN

    GVL_PHYSICAL_TRANSACTION.Cross_Actuator_Convergence_Skew := TRUE;

    L_Transaction_Valid := FALSE;
    L_Error_Code := 27000;
    L_Error_Text := 'Physical transaction epoch skew detected';
END_IF;

// Ordering race detection.
IF L_Transaction_Valid
AND GVL_PHYSICAL_TRANSACTION.Pump_Valve_Ordering_Race_Detected THEN
    L_Transaction_Valid := FALSE;
    L_Error_Code := 27001;
    L_Error_Text := 'Pump/valve ordering race detected';
END_IF;

// Brownout / rollback protection.
IF L_Transaction_Valid
AND GVL_PHYSICAL_TRANSACTION.Distributed_Actuator_Rollback_Detected THEN
    L_Transaction_Valid := FALSE;
    L_Error_Code := 27002;
    L_Error_Text := 'Distributed actuator rollback detected';
END_IF;

IF L_Transaction_Valid
AND GVL_PHYSICAL_TRANSACTION.Brownout_Partial_Switching_Detected THEN
    L_Transaction_Valid := FALSE;
    L_Error_Code := 27003;
    L_Error_Text := 'Brownout partial switching detected';
END_IF;

IF L_Transaction_Valid
AND GVL_PHYSICAL_TRANSACTION.Transaction_Timeout_Detected THEN
    L_Transaction_Valid := FALSE;
    L_Error_Code := 27004;
    L_Error_Text := 'Physical transaction timeout detected';
END_IF;

IF L_Transaction_Valid
AND GVL_PHYSICAL_TRANSACTION.Partial_Plant_Transition_Detected THEN
    L_Transaction_Valid := FALSE;
    L_Error_Code := 27005;
    L_Error_Text := 'Partial plant transition detected';
END_IF;

// All actuator transitions required.
IF L_Transaction_Valid
AND NOT GVL_PHYSICAL_TRANSACTION.Valve_Transition_Confirmed THEN
    L_Transaction_Valid := FALSE;
    L_Error_Code := 27010;
    L_Error_Text := 'Valve transition confirmation missing';
END_IF;

IF L_Transaction_Valid
AND NOT GVL_PHYSICAL_TRANSACTION.Pump_Transition_Confirmed THEN
    L_Transaction_Valid := FALSE;
    L_Error_Code := 27011;
    L_Error_Text := 'Pump transition confirmation missing';
END_IF;

IF L_Transaction_Valid
AND NOT GVL_PHYSICAL_TRANSACTION.Damper_Transition_Confirmed THEN
    L_Transaction_Valid := FALSE;
    L_Error_Code := 27012;
    L_Error_Text := 'Damper transition confirmation missing';
END_IF;

IF L_Transaction_Valid
AND NOT GVL_PHYSICAL_TRANSACTION.Relay_Bank_Transition_Confirmed THEN
    L_Transaction_Valid := FALSE;
    L_Error_Code := 27013;
    L_Error_Text := 'Relay bank transition confirmation missing';
END_IF;

// Stable plant convergence required.
IF L_Transaction_Valid
AND NOT GVL_PHYSICAL_TRANSACTION.Flow_Stabilization_Confirmed THEN
    L_Transaction_Valid := FALSE;
    L_Error_Code := 27020;
    L_Error_Text := 'Flow stabilization missing';
END_IF;

IF L_Transaction_Valid
AND NOT GVL_PHYSICAL_TRANSACTION.Pressure_Stabilization_Confirmed THEN
    L_Transaction_Valid := FALSE;
    L_Error_Code := 27021;
    L_Error_Text := 'Pressure stabilization missing';
END_IF;

IF L_Transaction_Valid
AND NOT GVL_PHYSICAL_TRANSACTION.Thermal_Response_Confirmed THEN
    L_Transaction_Valid := FALSE;
    L_Error_Code := 27022;
    L_Error_Text := 'Thermal response confirmation missing';
END_IF;

IF L_Transaction_Valid
AND NOT GVL_PHYSICAL_TRANSACTION.Electrical_Load_Stabilized THEN
    L_Transaction_Valid := FALSE;
    L_Error_Code := 27023;
    L_Error_Text := 'Electrical load stabilization missing';
END_IF;

IF L_Transaction_Valid THEN
    GVL_PHYSICAL_TRANSACTION.Physical_Transaction_Valid := TRUE;
    GVL_PHYSICAL_TRANSACTION.Physical_Transaction_Granted := TRUE;
    GVL_PHYSICAL_TRANSACTION.Physical_Transaction_Quarantine_Active := FALSE;

    GVL_PHYSICAL_TRANSACTION.All_Actuators_Converged := TRUE;
    GVL_PHYSICAL_TRANSACTION.Cross_Actuator_Epoch_Coherent := TRUE;
    GVL_PHYSICAL_TRANSACTION.Distributed_Actuation_Coherent := TRUE;
    GVL_PHYSICAL_TRANSACTION.Stable_Plant_State_Confirmed := TRUE;

    GVL_PHYSICAL_TRANSACTION.Physical_Transaction_Epoch :=
        GVL_PHYSICAL_TRANSACTION.Physical_Transaction_Command_Epoch;

    GVL_PHYSICAL_TRANSACTION.Physical_Transaction_Last_Update_MS :=
        L_Now_MS;

    GVL_PHYSICAL_TRANSACTION.Physical_Transaction_Lease_Expired := FALSE;

    GVL_PHYSICAL_TRANSACTION.Physical_Transaction_Last_Error_Code := 0;
    GVL_PHYSICAL_TRANSACTION.Physical_Transaction_Last_Error_Text := '';
ELSE
    GVL_PHYSICAL_TRANSACTION.Physical_Transaction_Valid := FALSE;
    GVL_PHYSICAL_TRANSACTION.Physical_Transaction_Granted := FALSE;
    GVL_PHYSICAL_TRANSACTION.Physical_Transaction_Quarantine_Active := TRUE;

    GVL_PHYSICAL_TRANSACTION.Physical_Transaction_Lease_Expired := TRUE;

    GVL_PHYSICAL_TRANSACTION.Physical_Transaction_Last_Error_Code :=
        L_Error_Code;

    GVL_PHYSICAL_TRANSACTION.Physical_Transaction_Last_Error_Text :=
        L_Error_Text;

    GVL_PHYSICAL_TRANSACTION.Physical_Transaction_Invalidation_Count :=
        GVL_PHYSICAL_TRANSACTION.Physical_Transaction_Invalidation_Count + 1;
END_IF;

END_PROGRAM

(* ---- PRG_PLC_Fencing_Governor.st ---- *)
PROGRAM PRG_PLC_Fencing_Governor
VAR
    L_Now_MS : UDINT;
    L_Delta_MS : UDINT;
    L_Authority_Valid : BOOL := TRUE;
    L_Error_Code : UDINT := 0;
    L_Error_Text : STRING(160) := '';
END_VAR

L_Now_MS := GVL_STATUS.G_System_Time_MS;
L_Authority_Valid := TRUE;
L_Error_Code := 0;
L_Error_Text := '';

// ======================================================
// PLC FENCING GOVERNOR
// ======================================================
// Governs distributed PLC ownership semantics.
// Prevents stale-owner resurrection and split-brain.
// ======================================================

GVL_PLC_FENCING.PLC_Split_Brain_Detected := FALSE;
GVL_PLC_FENCING.PLC_Stale_Owner_Detected := FALSE;
GVL_PLC_FENCING.PLC_Asymmetric_Partition_Detected := FALSE;
GVL_PLC_FENCING.PLC_Forced_Safe_Quarantine := FALSE;

// Active PLC ownership validation.
IF L_Authority_Valid AND (NOT GVL_STATUS.G_Is_Active_PLC) THEN
    L_Authority_Valid := FALSE;
    L_Error_Code := 7001;
    L_Error_Text := 'PLC ownership inactive';
END_IF;

// Lease freshness validation.
L_Delta_MS := L_Now_MS - GVL_PLC_FENCING.PLC_Last_Lease_Refresh_MS;

IF L_Authority_Valid AND GVL_PLC_FENCING.PLC_Lease_Active THEN
    IF L_Delta_MS > GVL_PLC_FENCING.PLC_Lease_Timeout_MS THEN
        L_Authority_Valid := FALSE;
        L_Error_Code := 7002;
        L_Error_Text := 'PLC lease expired';
    END_IF;
END_IF;

// Heartbeat-only ownership is unsafe.
IF L_Authority_Valid AND GVL_PLC_FENCING.PLC_Heartbeat_Only_Mode THEN
    L_Authority_Valid := FALSE;
    L_Error_Code := 7003;
    L_Error_Text := 'Heartbeat-only ownership rejected';
END_IF;

// Publish authoritative fencing state.
IF L_Authority_Valid THEN
    GVL_PLC_FENCING.PLC_Ownership_Epoch := GVL_PLC_FENCING.PLC_Ownership_Epoch + 1;
    GVL_PLC_FENCING.PLC_Fencing_Token := GVL_PLC_FENCING.PLC_Ownership_Epoch;

    GVL_PLC_FENCING.PLC_Ownership_Valid := TRUE;
    GVL_PLC_FENCING.PLC_Semantic_Authority_Valid := TRUE;

    GVL_PLC_FENCING.PLC_Lease_Active := TRUE;
    GVL_PLC_FENCING.PLC_Lease_Expired := FALSE;

    GVL_PLC_FENCING.PLC_Last_Lease_Refresh_MS := L_Now_MS;
    GVL_PLC_FENCING.PLC_Last_Authority_Validation_MS := L_Now_MS;

    GVL_PLC_FENCING.PLC_Last_Error_Code := 0;
    GVL_PLC_FENCING.PLC_Last_Error_Text := '';
ELSE
    GVL_PLC_FENCING.PLC_Ownership_Valid := FALSE;
    GVL_PLC_FENCING.PLC_Semantic_Authority_Valid := FALSE;

    GVL_PLC_FENCING.PLC_Lease_Expired := TRUE;
    GVL_PLC_FENCING.PLC_Forced_Safe_Quarantine := TRUE;

    GVL_PLC_FENCING.PLC_Last_Error_Code := L_Error_Code;
    GVL_PLC_FENCING.PLC_Last_Error_Text := L_Error_Text;

    IF L_Error_Code = 7002 THEN
        GVL_PLC_FENCING.PLC_Stale_Owner_Detected := TRUE;
    END_IF;

    IF L_Error_Code = 7003 THEN
        GVL_PLC_FENCING.PLC_Split_Brain_Detected := TRUE;
        GVL_PLC_FENCING.PLC_Asymmetric_Partition_Detected := TRUE;
    END_IF;

    GVL_PLC_FENCING.PLC_Fencing_Invalidation_Count := GVL_PLC_FENCING.PLC_Fencing_Invalidation_Count + 1;
END_IF;
END_PROGRAM

(* ---- PRG_Policy.st ---- *)
PROGRAM PRG_Policy

// ============================================================
// CONFIGURATION SAFETY CLAMP
// ============================================================
// Configuration validation is diagnostic-only here.
// System mode ownership remains in FB_State_Manager via
// FB_System_Health_Orchestrator. Policy must not directly write
// GVL_STATE.G_System_Mode.
IF GVL_CONFIG_VALIDATION.G_Config_Force_Safe_Mode AND
   (NOT GVL_CONFIG_VALIDATION.G_Config_Valid) AND
   (GVL_STATE.G_System_Mode = E_System_Operating_Mode.MODE_NORMAL) THEN
    GVL_STATUS.G_Diagnostics.Subsystem_Degraded := TRUE;
    GVL_STATUS.G_System_Mode_Text := 'CONFIG DEGRADED';
END_IF;

// ============================================================
// SCENARIO POLICY OWNER
// ============================================================

// 1. Base priority resolution
IF GVL_STATE.G_System_Mode = E_System_Operating_Mode.MODE_SAFE_STOP THEN
    GVL_POLICY.G_Scenario_Intent := E_SCENARIO_TYPE.SCENARIO_NONE;
    GVL_POLICY.G_Scenario_Source := SRC_SAFETY;

ELSIF GVL_POLICY.G_Scenario_Request_Operator <> E_SCENARIO_TYPE.SCENARIO_NONE THEN
    GVL_POLICY.G_Scenario_Intent := GVL_POLICY.G_Scenario_Request_Operator;
    GVL_POLICY.G_Scenario_Source := SRC_OPERATOR;

ELSIF GVL_POLICY.G_Scenario_Request_Gateway <> E_SCENARIO_TYPE.SCENARIO_NONE THEN
    GVL_POLICY.G_Scenario_Intent := GVL_POLICY.G_Scenario_Request_Gateway;
    GVL_POLICY.G_Scenario_Source := SRC_GATEWAY;

ELSIF GVL_POLICY.G_Scenario_Request_Rule <> E_SCENARIO_TYPE.SCENARIO_NONE THEN
    GVL_POLICY.G_Scenario_Intent := GVL_POLICY.G_Scenario_Request_Rule;
    GVL_POLICY.G_Scenario_Source := SRC_RULE;

ELSE
    GVL_POLICY.G_Scenario_Intent := GVL_STATUS.G_Current_Scenario;
    GVL_POLICY.G_Scenario_Source := SRC_NONE;
END_IF;

// 2. Fail-safe clamp
CASE GVL_STATE.G_System_Mode OF
    E_System_Operating_Mode.MODE_SAFE_STOP:
        GVL_POLICY.G_Scenario_Intent := E_SCENARIO_TYPE.SCENARIO_NONE;
        GVL_POLICY.G_Scenario_Source := SRC_SAFETY;

    E_System_Operating_Mode.MODE_FREEZE_PROTECTION:
        GVL_POLICY.G_Scenario_Intent := E_SCENARIO_TYPE.SCENARIO_NONE;
        GVL_POLICY.G_Scenario_Source := SRC_POLICY;

    E_System_Operating_Mode.MODE_DEGRADED:
        CASE GVL_POLICY.G_Scenario_Intent OF
            E_SCENARIO_TYPE.SCENARIO_NONE,
            E_SCENARIO_TYPE.SCENARIO_PRESENCE,
            E_SCENARIO_TYPE.SCENARIO_AWAY,
            E_SCENARIO_TYPE.SCENARIO_SLEEP:
                ;
        ELSE
            GVL_POLICY.G_Scenario_Intent := E_SCENARIO_TYPE.SCENARIO_NONE;
            GVL_POLICY.G_Scenario_Source := SRC_POLICY;
        END_CASE;
END_CASE;

// 3. Context automation
IF GVL_STATE.G_System_Mode = E_System_Operating_Mode.MODE_NORMAL THEN
    IF GVL_ALARM.G_Security_Armed AND
       (GVL_POLICY.G_Scenario_Request_Operator = E_SCENARIO_TYPE.SCENARIO_NONE) AND
       (GVL_POLICY.G_Scenario_Request_Gateway = E_SCENARIO_TYPE.SCENARIO_NONE) AND
       (GVL_POLICY.G_Scenario_Request_Rule = E_SCENARIO_TYPE.SCENARIO_NONE) AND
       (GVL_POLICY.G_Scenario_Intent <> E_SCENARIO_TYPE.SCENARIO_AWAY) THEN
        GVL_POLICY.G_Scenario_Intent := E_SCENARIO_TYPE.SCENARIO_AWAY;
        GVL_POLICY.G_Scenario_Source := SRC_POLICY;
    END_IF;
END_IF;

// 4. Degraded adaptation
IF GVL_STATE.G_System_Mode = E_System_Operating_Mode.MODE_DEGRADED THEN
    IF (GVL_POLICY.G_Scenario_Request_Operator = E_SCENARIO_TYPE.SCENARIO_NONE) AND
       (GVL_POLICY.G_Scenario_Request_Gateway = E_SCENARIO_TYPE.SCENARIO_NONE) AND
       (GVL_POLICY.G_Scenario_Request_Rule = E_SCENARIO_TYPE.SCENARIO_NONE) THEN

        IF GVL_ALARM.G_Security_Armed THEN
            GVL_POLICY.G_Scenario_Intent := E_SCENARIO_TYPE.SCENARIO_AWAY;
            GVL_POLICY.G_Scenario_Source := SRC_POLICY;

        ELSIF GVL_POLICY.G_Scenario_Intent = E_SCENARIO_TYPE.SCENARIO_PRESENCE THEN
            GVL_POLICY.G_Scenario_Intent := E_SCENARIO_TYPE.SCENARIO_SLEEP;
            GVL_POLICY.G_Scenario_Source := SRC_POLICY;
        END_IF;
    END_IF;
END_IF;

// 5. Heating bridge
GVL_STATE.G_Preheat_Request := GVL_POLICY.G_Rule_Preheat_Request;
GVL_STATE.G_Freeze_Request :=
    (GVL_STATE.G_System_Mode = E_System_Operating_Mode.MODE_FREEZE_PROTECTION);
END_PROGRAM

(* ---- PRG_Proof_Continuity_Audit_Governor.st ---- *)
PROGRAM PRG_Proof_Continuity_Audit_Governor
// PASSIVE PROOF AUDIT ONLY

GVL_PROOF_CONTINUITY_AUDIT_FABRIC.Proof_Continuity_Observed :=
    GVL_SEMANTIC_DRIFT_OBSERVABILITY_FABRIC.Semantic_Continuity_Observed;

GVL_PROOF_CONTINUITY_AUDIT_FABRIC.Proof_Lineage_Coherent := TRUE;
GVL_PROOF_CONTINUITY_AUDIT_FABRIC.Proof_Historical_Integrity_Observed := TRUE;

END_PROGRAM

(* ---- PRG_Recovery_Cleanup_Governor.st ---- *)
PROGRAM PRG_Recovery_Cleanup_Governor
VAR
    L_Now_MS : UDINT;
    L_Recovery_Valid : BOOL := TRUE;
    L_Error_Code : UDINT := 0;
    L_Error_Text : STRING(160) := '';

    L_Distributed_Recovery_Allowed : BOOL;
    L_Cluster_Recovery_Lock : BOOL;
    L_Cluster_Quarantine : BOOL;

    L_Finalized_Publication_Continuity : BOOL;
END_VAR

L_Now_MS := GVL_STATUS.G_System_Time_MS;
L_Recovery_Valid := TRUE;
L_Error_Code := 0;
L_Error_Text := '';

GVL_RECOVERY_GOVERNANCE.Recovery_Semantic_Residue_Detected := FALSE;
GVL_RECOVERY_GOVERNANCE.Recovery_Degraded_State_Residual := FALSE;
GVL_RECOVERY_GOVERNANCE.Recovery_Retained_State_Residual := FALSE;

L_Distributed_Recovery_Allowed :=
    GVL_Distributed_Execution_Gates.G_Can_Recover;

L_Cluster_Recovery_Lock :=
    GVL_Cluster_Runtime_FSM.G_State_Recovery_Lock;

L_Cluster_Quarantine :=
    GVL_Cluster_Runtime_FSM.G_State_Quarantine;

// Finalized publication continuity.
L_Finalized_Publication_Continuity :=
    GVL_DISTRIBUTED_SNAPSHOT.Distributed_Publication_Reconciled
    AND GVL_DISTRIBUTED_SNAPSHOT.Distributed_Publication_Freeze_Valid
    AND GVL_DISTRIBUTED_SNAPSHOT.Distributed_Snapshot_Consistent
    AND GVL_DISTRIBUTED_COMMIT.Distributed_Commit_Valid
    AND NOT GVL_DISTRIBUTED_COMMIT.Commit_Lease_Expired
    AND GVL_OUTPUT_EPOCH.Output_Publication_Valid
    AND GVL_OUTPUT_EPOCH.Output_Runtime_Epoch_Valid
    AND NOT GVL_OUTPUT_EPOCH.Output_Lease_Expired
    AND NOT GVL_OUTPUT_EPOCH.Output_Forced_Safe_Decay;

IF NOT GVL_TIME_MONOTONIC.Monotonic_Time_Valid THEN
    L_Recovery_Valid := FALSE;
    L_Error_Code := 9001;
    L_Error_Text := 'Recovery monotonic authority invalid';
END_IF;

IF L_Recovery_Valid
   AND NOT L_Distributed_Recovery_Allowed THEN

    L_Recovery_Valid := FALSE;

    L_Error_Code := 9010;
    L_Error_Text :=
        'Distributed recovery governance restricted';

END_IF;

IF L_Recovery_Valid
   AND L_Cluster_Recovery_Lock THEN

    L_Recovery_Valid := FALSE;

    L_Error_Code := 9011;
    L_Error_Text :=
        'Cluster recovery-lock active';

END_IF;

IF L_Recovery_Valid
   AND L_Cluster_Quarantine THEN

    L_Recovery_Valid := FALSE;

    L_Error_Code := 9012;
    L_Error_Text :=
        'Cluster quarantine active';

END_IF;

IF GVL_SAFETY_RECOVERY.G_Recovery_Active THEN
    GVL_RECOVERY_GOVERNANCE.Recovery_Quarantine_Active := TRUE;
    GVL_RECOVERY_GOVERNANCE.Recovery_Last_Cleanup_Start_MS := L_Now_MS;

    L_Recovery_Valid := FALSE;

    IF L_Error_Code = 0 THEN
        L_Error_Code := 9002;
        L_Error_Text := 'Recovery quarantine active';
    END_IF;
END_IF;

IF L_Recovery_Valid AND GVL_DEGRADED.G_System_Degraded THEN
    L_Recovery_Valid := FALSE;
    L_Error_Code := 9003;
    L_Error_Text := 'Residual degraded state detected';

    GVL_RECOVERY_GOVERNANCE.Recovery_Degraded_State_Residual := TRUE;
END_IF;

IF L_Recovery_Valid AND GVL_TIME_MONOTONIC.Retained_Time_Invalid THEN
    L_Recovery_Valid := FALSE;
    L_Error_Code := 9004;
    L_Error_Text := 'Retained state residue detected';

    GVL_RECOVERY_GOVERNANCE.Recovery_Retained_State_Residual := TRUE;
END_IF;

IF L_Recovery_Valid THEN
    GVL_RECOVERY_GOVERNANCE.Recovery_Epoch := GVL_RECOVERY_GOVERNANCE.Recovery_Epoch + 1;
    GVL_RECOVERY_GOVERNANCE.Recovery_Cleanup_Epoch := GVL_RECOVERY_GOVERNANCE.Recovery_Cleanup_Epoch + 1;

    GVL_RECOVERY_GOVERNANCE.Recovery_Governance_Valid := TRUE;

    // Cleanup release requires finalized publication continuity.
    IF GVL_CONVERGENCE.Convergence_Release_Allowed
       AND L_Finalized_Publication_Continuity THEN

        GVL_RECOVERY_GOVERNANCE.Recovery_Cleanup_Completed := TRUE;
        GVL_RECOVERY_GOVERNANCE.Recovery_Cleanup_Verified := TRUE;
        GVL_RECOVERY_GOVERNANCE.Recovery_Quarantine_Active := FALSE;
        GVL_RECOVERY_GOVERNANCE.Recovery_Forced_Safe_Mode := FALSE;
        GVL_RECOVERY_GOVERNANCE.Recovery_Last_Cleanup_End_MS := L_Now_MS;

        GVL_RECOVERY_GOVERNANCE.Recovery_Last_Error_Code := 0;
        GVL_RECOVERY_GOVERNANCE.Recovery_Last_Error_Text := '';
    ELSE
        GVL_RECOVERY_GOVERNANCE.Recovery_Cleanup_Completed := FALSE;
        GVL_RECOVERY_GOVERNANCE.Recovery_Cleanup_Verified := FALSE;
        GVL_RECOVERY_GOVERNANCE.Recovery_Quarantine_Active := TRUE;
        GVL_RECOVERY_GOVERNANCE.Recovery_Forced_Safe_Mode := TRUE;

        GVL_RECOVERY_GOVERNANCE.Recovery_Last_Error_Code := 9005;
        GVL_RECOVERY_GOVERNANCE.Recovery_Last_Error_Text := 'Recovery cleanup waiting for finalized publication continuity';
    END_IF;
ELSE
    GVL_RECOVERY_GOVERNANCE.Recovery_Governance_Valid := FALSE;
    GVL_RECOVERY_GOVERNANCE.Recovery_Cleanup_Completed := FALSE;
    GVL_RECOVERY_GOVERNANCE.Recovery_Cleanup_Verified := FALSE;

    GVL_RECOVERY_GOVERNANCE.Recovery_Semantic_Residue_Detected := TRUE;
    GVL_RECOVERY_GOVERNANCE.Recovery_Forced_Safe_Mode := TRUE;

    GVL_RECOVERY_GOVERNANCE.Recovery_Last_Error_Code := L_Error_Code;
    GVL_RECOVERY_GOVERNANCE.Recovery_Last_Error_Text := L_Error_Text;

    GVL_RECOVERY_GOVERNANCE.Recovery_Invalidation_Count := GVL_RECOVERY_GOVERNANCE.Recovery_Invalidation_Count + 1;
END_IF;
END_PROGRAM

(* ---- PRG_Residual_Energy_State_Governor.st ---- *)
PROGRAM PRG_Residual_Energy_State_Governor
IF GVL_ENERGY_ISOLATION_CAUSALITY_FABRIC.Energy_Isolation_Causality_Granted
AND NOT GVL_RESIDUAL_ENERGY_STATE_FABRIC.Latent_Unsafe_Actuation_Detected
AND NOT GVL_RESIDUAL_ENERGY_STATE_FABRIC.Residual_Energy_Persistence_Detected
AND NOT GVL_RESIDUAL_ENERGY_STATE_FABRIC.Unsafe_Thermal_Energy_Retention THEN

    GVL_RESIDUAL_ENERGY_STATE_FABRIC.Residual_Energy_State_Valid := TRUE;
    GVL_RESIDUAL_ENERGY_STATE_FABRIC.Residual_Energy_Bounded := TRUE;
    GVL_RESIDUAL_ENERGY_STATE_FABRIC.Residual_Actuation_Energy_Safe := TRUE;
    GVL_RESIDUAL_ENERGY_STATE_FABRIC.Thermal_Energy_Dissipation_Stable := TRUE;
END_IF;
END_PROGRAM

(* ---- PRG_Runtime_Budget_Governor.st ---- *)
PROGRAM PRG_Runtime_Budget_Governor
// RUNTIME BUDGET ENFORCEMENT
// READ-ONLY / NON-INVASIVE

GVL_RUNTIME_BUDGET_ENFORCEMENT.Runtime_Budget_Pressure_Observed :=
    GVL_CANONICAL_RUNTIME_FABRIC_REGISTRY.Runtime_Complexity_Pressure_Observed;

GVL_RUNTIME_BUDGET_ENFORCEMENT.Governance_Runtime_Overhead_Observed :=
    GVL_CANONICAL_RUNTIME_FABRIC_REGISTRY.Governance_Runtime_Cost_Observed;

GVL_RUNTIME_BUDGET_ENFORCEMENT.Verification_Runtime_Budget_Observed :=
    GVL_CANONICAL_RUNTIME_FABRIC_REGISTRY.Verification_Chaining_Limit_Reached;

GVL_RUNTIME_BUDGET_ENFORCEMENT.Observability_Runtime_Budget_Observed :=
    GVL_CANONICAL_RUNTIME_FABRIC_REGISTRY.Observability_Amplification_Limit_Reached;

IF GVL_RUNTIME_BUDGET_ENFORCEMENT.Runtime_Budget_Pressure_Observed THEN
    GVL_RUNTIME_BUDGET_ENFORCEMENT.Runtime_Stability_Budget_At_Risk := TRUE;
END_IF;

IF GVL_RUNTIME_BUDGET_ENFORCEMENT.Verification_Runtime_Budget_Observed THEN
    GVL_RUNTIME_BUDGET_ENFORCEMENT.Verification_Time_Budget_Exceeded := TRUE;
    GVL_RUNTIME_BUDGET_ENFORCEMENT.Verification_Induced_Runtime_Risk := TRUE;
END_IF;

IF GVL_RUNTIME_BUDGET_ENFORCEMENT.Observability_Runtime_Budget_Observed THEN
    GVL_RUNTIME_BUDGET_ENFORCEMENT.Observability_Amplification_Budget_Exceeded := TRUE;
END_IF;

END_PROGRAM

(* ---- PRG_Runtime_Compression_Governor.st ---- *)
PROGRAM PRG_Runtime_Compression_Governor
// ARCHITECTURAL CONSOLIDATION & RUNTIME COMPRESSION
// READ-ONLY / NON-INVASIVE

GVL_CANONICAL_RUNTIME_FABRIC_REGISTRY.Runtime_Complexity_Pressure_Observed :=
    GVL_SURVIVABILITY_INTELLIGENCE_FABRIC.Governance_Saturation_Pressure_Observed;

GVL_CANONICAL_RUNTIME_FABRIC_REGISTRY.Governance_Runtime_Cost_Observed :=
    GVL_OPERATIONAL_INTELLIGENCE_FABRIC.Governance_Complexity_Pressure_Observed;

GVL_CANONICAL_RUNTIME_FABRIC_REGISTRY.Verification_Induced_Instability_Risk :=
    GVL_SURVIVABILITY_INTELLIGENCE_FABRIC.Chronic_Degradation_Risk_Increasing;

IF GVL_OPERATIONAL_INTELLIGENCE_FABRIC.Governance_Saturation_Observed THEN
    GVL_CANONICAL_RUNTIME_FABRIC_REGISTRY.Governance_Scattering_Observed := TRUE;
    GVL_CANONICAL_RUNTIME_FABRIC_REGISTRY.Semantic_Duplication_Observed := TRUE;
END_IF;

IF GVL_CANONICAL_RUNTIME_FABRIC_REGISTRY.Runtime_Complexity_Pressure_Observed THEN
    GVL_CANONICAL_RUNTIME_FABRIC_REGISTRY.Governance_Depth_Limit_Reached := TRUE;
END_IF;

IF GVL_CANONICAL_RUNTIME_FABRIC_REGISTRY.Governance_Runtime_Cost_Observed THEN
    GVL_CANONICAL_RUNTIME_FABRIC_REGISTRY.Verification_Chaining_Limit_Reached := TRUE;
END_IF;

IF GVL_OPERATIONAL_INTELLIGENCE_FABRIC.Operational_Opacity_Observed THEN
    GVL_CANONICAL_RUNTIME_FABRIC_REGISTRY.Observability_Amplification_Limit_Reached := TRUE;
END_IF;

END_PROGRAM

(* ---- PRG_Runtime_Resource_Authority_Governor.st ---- *)
PROGRAM PRG_Runtime_Resource_Authority_Governor
VAR
    L_Now_MS : UDINT;
    L_Runtime_Valid : BOOL := TRUE;
    L_Error_Code : UDINT := 0;
    L_Error_Text : STRING(160) := '';
END_VAR

L_Now_MS := GVL_STATUS.G_System_Time_MS;
L_Runtime_Valid := TRUE;
L_Error_Code := 0;
L_Error_Text := '';

// Fail-safe defaults.
GVL_RUNTIME_RESOURCE_AUTHORITY.Runtime_Resource_Authority_Valid := FALSE;
GVL_RUNTIME_RESOURCE_AUTHORITY.Runtime_Resource_Authority_Granted := FALSE;
GVL_RUNTIME_RESOURCE_AUTHORITY.Runtime_Resource_Quarantine_Active := TRUE;

GVL_RUNTIME_RESOURCE_AUTHORITY.Deterministic_Cycle_Time_Valid := FALSE;
GVL_RUNTIME_RESOURCE_AUTHORITY.Task_Jitter_Within_Bounds := FALSE;
GVL_RUNTIME_RESOURCE_AUTHORITY.Watchdog_Margin_Stable := FALSE;
GVL_RUNTIME_RESOURCE_AUTHORITY.Runtime_Latency_Stable := FALSE;
GVL_RUNTIME_RESOURCE_AUTHORITY.Queue_Backlog_Stable := FALSE;

// Environmental authority required.
IF NOT GVL_ENVIRONMENTAL_AUTHORITY.Environmental_Authority_Granted THEN
    L_Runtime_Valid := FALSE;
    L_Error_Code := 30000;
    L_Error_Text := 'Environmental authority not granted';
END_IF;

// Resource exhaustion detectors.
IF GVL_RUNTIME_RESOURCE_AUTHORITY.Hidden_Jitter_Amplification_Detected THEN
    L_Runtime_Valid := FALSE;
    L_Error_Code := 30001;
    L_Error_Text := 'Hidden jitter amplification detected';
END_IF;

IF GVL_RUNTIME_RESOURCE_AUTHORITY.Queue_Induced_Authority_Lag_Detected THEN
    L_Runtime_Valid := FALSE;
    L_Error_Code := 30002;
    L_Error_Text := 'Queue-induced authority lag detected';
END_IF;

IF GVL_RUNTIME_RESOURCE_AUTHORITY.Watchdog_Near_Death_Oscillation_Detected THEN
    L_Runtime_Valid := FALSE;
    L_Error_Code := 30003;
    L_Error_Text := 'Watchdog near-death oscillation detected';
END_IF;

IF GVL_RUNTIME_RESOURCE_AUTHORITY.Runtime_Starvation_Race_Detected THEN
    L_Runtime_Valid := FALSE;
    L_Error_Code := 30004;
    L_Error_Text := 'Runtime starvation race detected';
END_IF;

IF GVL_RUNTIME_RESOURCE_AUTHORITY.Cycle_Collapse_SplitBrain_Detected THEN
    L_Runtime_Valid := FALSE;
    L_Error_Code := 30005;
    L_Error_Text := 'Cycle collapse split-brain detected';
END_IF;

IF GVL_RUNTIME_RESOURCE_AUTHORITY.Heap_Fragmentation_Critical THEN
    L_Runtime_Valid := FALSE;
    L_Error_Code := 30006;
    L_Error_Text := 'Critical heap fragmentation detected';
END_IF;

IF GVL_RUNTIME_RESOURCE_AUTHORITY.Fieldbus_Backlog_Saturation_Detected THEN
    L_Runtime_Valid := FALSE;
    L_Error_Code := 30007;
    L_Error_Text := 'Fieldbus backlog saturation detected';
END_IF;

// Deterministic execution envelope validation.
IF L_Runtime_Valid
AND (GVL_RUNTIME_RESOURCE_AUTHORITY.Current_Task_Jitter_US >
     GVL_RUNTIME_RESOURCE_AUTHORITY.Max_Allowed_Task_Jitter_US) THEN

    L_Runtime_Valid := FALSE;
    L_Error_Code := 30010;
    L_Error_Text := 'Task jitter exceeds deterministic envelope';
END_IF;

IF L_Runtime_Valid
AND (GVL_RUNTIME_RESOURCE_AUTHORITY.Current_Runtime_Latency_US >
     GVL_RUNTIME_RESOURCE_AUTHORITY.Max_Allowed_Runtime_Latency_US) THEN

    L_Runtime_Valid := FALSE;
    L_Error_Code := 30011;
    L_Error_Text := 'Runtime latency exceeds deterministic envelope';
END_IF;

IF L_Runtime_Valid
AND (GVL_RUNTIME_RESOURCE_AUTHORITY.Current_Fieldbus_Queue_Depth >
     GVL_RUNTIME_RESOURCE_AUTHORITY.Max_Allowed_Fieldbus_Queue_Depth) THEN

    L_Runtime_Valid := FALSE;
    L_Error_Code := 30012;
    L_Error_Text := 'Fieldbus queue depth exceeds deterministic envelope';
END_IF;

IF L_Runtime_Valid
AND (GVL_RUNTIME_RESOURCE_AUTHORITY.Current_Watchdog_Margin_MS <
     GVL_RUNTIME_RESOURCE_AUTHORITY.Minimum_Watchdog_Margin_MS) THEN

    L_Runtime_Valid := FALSE;
    L_Error_Code := 30013;
    L_Error_Text := 'Watchdog margin below deterministic envelope';
END_IF;

IF L_Runtime_Valid THEN
    GVL_RUNTIME_RESOURCE_AUTHORITY.Runtime_Resource_Authority_Valid := TRUE;
    GVL_RUNTIME_RESOURCE_AUTHORITY.Runtime_Resource_Authority_Granted := TRUE;
    GVL_RUNTIME_RESOURCE_AUTHORITY.Runtime_Resource_Quarantine_Active := FALSE;

    GVL_RUNTIME_RESOURCE_AUTHORITY.Deterministic_Cycle_Time_Valid := TRUE;
    GVL_RUNTIME_RESOURCE_AUTHORITY.Task_Jitter_Within_Bounds := TRUE;
    GVL_RUNTIME_RESOURCE_AUTHORITY.Watchdog_Margin_Stable := TRUE;
    GVL_RUNTIME_RESOURCE_AUTHORITY.Runtime_Latency_Stable := TRUE;
    GVL_RUNTIME_RESOURCE_AUTHORITY.Queue_Backlog_Stable := TRUE;

    GVL_RUNTIME_RESOURCE_AUTHORITY.Runtime_Resource_Authority_Epoch :=
        GVL_ENVIRONMENTAL_AUTHORITY.Environmental_Authority_Epoch;

    GVL_RUNTIME_RESOURCE_AUTHORITY.Runtime_Resource_Authority_Epoch_Coherent := TRUE;

    GVL_RUNTIME_RESOURCE_AUTHORITY.Runtime_Resource_Last_Update_MS :=
        L_Now_MS;

    GVL_RUNTIME_RESOURCE_AUTHORITY.Runtime_Resource_Lease_Expired := FALSE;

    GVL_RUNTIME_RESOURCE_AUTHORITY.Runtime_Resource_Last_Error_Code := 0;
    GVL_RUNTIME_RESOURCE_AUTHORITY.Runtime_Resource_Last_Error_Text := '';
ELSE
    GVL_RUNTIME_RESOURCE_AUTHORITY.Runtime_Resource_Authority_Valid := FALSE;
    GVL_RUNTIME_RESOURCE_AUTHORITY.Runtime_Resource_Authority_Granted := FALSE;
    GVL_RUNTIME_RESOURCE_AUTHORITY.Runtime_Resource_Quarantine_Active := TRUE;

    GVL_RUNTIME_RESOURCE_AUTHORITY.Runtime_Resource_Lease_Expired := TRUE;

    GVL_RUNTIME_RESOURCE_AUTHORITY.Runtime_Resource_Last_Error_Code :=
        L_Error_Code;

    GVL_RUNTIME_RESOURCE_AUTHORITY.Runtime_Resource_Last_Error_Text :=
        L_Error_Text;

    GVL_RUNTIME_RESOURCE_AUTHORITY.Runtime_Resource_Invalidation_Count :=
        GVL_RUNTIME_RESOURCE_AUTHORITY.Runtime_Resource_Invalidation_Count + 1;
END_IF;

END_PROGRAM

(* ---- PRG_Runtime_Snapshot_Governor.st ---- *)
PROGRAM PRG_Runtime_Snapshot_Governor
VAR
    L_Now_MS : UDINT;
    L_Snapshot_Valid : BOOL := TRUE;
    L_Error_Code : UDINT := 0;
    L_Error_Text : STRING(160) := '';

    L_Distributed_Publication_Healthy : BOOL;
END_VAR

L_Now_MS := GVL_STATUS.G_System_Time_MS;
L_Snapshot_Valid := TRUE;
L_Error_Code := 0;
L_Error_Text := '';

// ======================================================
// IMMUTABLE RUNTIME SNAPSHOT GOVERNOR
// ======================================================
// Governs immutable publication snapshot semantics.
// Prevents mutable runtime publication leakage.
//
// Runtime snapshot is upstream of output freshness.
// However distributed publication continuity must
// still remain semantically consistent.
// ======================================================

GVL_RUNTIME_SNAPSHOT.Snapshot_Mutation_Detected := FALSE;
GVL_RUNTIME_SNAPSHOT.Snapshot_Publication_Allowed := FALSE;
GVL_RUNTIME_SNAPSHOT.Snapshot_Frozen := FALSE;

// ------------------------------------------------------
// Runtime authority linkage.
// ------------------------------------------------------

IF NOT GVL_RUNTIME_EPOCH.Runtime_Runtime_Barrier_OK THEN
    L_Snapshot_Valid := FALSE;
    L_Error_Code := 12000;
    L_Error_Text := 'Runtime authority invalid';
END_IF;

// ------------------------------------------------------
// Distributed publication continuity linkage.
// ------------------------------------------------------

L_Distributed_Publication_Healthy :=
    GVL_DISTRIBUTED_SNAPSHOT.Distributed_Publication_Reconciled
    AND GVL_DISTRIBUTED_SNAPSHOT.Distributed_Publication_Freeze_Valid
    AND GVL_DISTRIBUTED_SNAPSHOT.Distributed_Snapshot_Consistent
    AND GVL_DISTRIBUTED_COMMIT.Distributed_Commit_Valid
    AND GVL_DISTRIBUTED_COMMIT.Publication_Prepare_Valid
    AND GVL_DISTRIBUTED_COMMIT.Publication_Commit_Confirmed
    AND NOT GVL_DISTRIBUTED_COMMIT.Peer_Commit_Mismatch
    AND NOT GVL_DISTRIBUTED_COMMIT.Commit_Lease_Expired;

IF L_Snapshot_Valid
AND NOT L_Distributed_Publication_Healthy
THEN
    L_Snapshot_Valid := FALSE;
    L_Error_Code := 12001;
    L_Error_Text := 'Distributed publication continuity invalid';
END_IF;

// ------------------------------------------------------
// Mutation detection foundation.
// ------------------------------------------------------

IF L_Snapshot_Valid
AND GVL_RUNTIME_EPOCH.Runtime_Impossible_State_Detected
THEN
    L_Snapshot_Valid := FALSE;
    L_Error_Code := 12003;
    L_Error_Text := 'Runtime mutation anomaly detected';

    GVL_RUNTIME_SNAPSHOT.Snapshot_Mutation_Detected := TRUE;
END_IF;

// ------------------------------------------------------
// Immutable snapshot freeze semantics.
// ------------------------------------------------------

IF L_Snapshot_Valid THEN
    GVL_RUNTIME_SNAPSHOT.Snapshot_Frozen := TRUE;
    GVL_RUNTIME_SNAPSHOT.Snapshot_Publication_Allowed := TRUE;

    GVL_RUNTIME_SNAPSHOT.Snapshot_Copy_Valid := TRUE;
    GVL_RUNTIME_SNAPSHOT.Snapshot_Isolation_Valid := TRUE;

    GVL_RUNTIME_SNAPSHOT.Snapshot_Runtime_Authority_Valid := TRUE;

    GVL_RUNTIME_SNAPSHOT.Snapshot_Freeze_Start_MS := L_Now_MS;
    GVL_RUNTIME_SNAPSHOT.Snapshot_Last_Publication_MS := L_Now_MS;

    GVL_RUNTIME_SNAPSHOT.Snapshot_Epoch := GVL_RUNTIME_SNAPSHOT.Snapshot_Epoch + 1;
    GVL_RUNTIME_SNAPSHOT.Snapshot_Publication_Epoch := GVL_RUNTIME_SNAPSHOT.Snapshot_Publication_Epoch + 1;

    GVL_RUNTIME_SNAPSHOT.Snapshot_Last_Error_Code := 0;
    GVL_RUNTIME_SNAPSHOT.Snapshot_Last_Error_Text := '';
ELSE
    GVL_RUNTIME_SNAPSHOT.Snapshot_Frozen := FALSE;
    GVL_RUNTIME_SNAPSHOT.Snapshot_Publication_Allowed := FALSE;

    GVL_RUNTIME_SNAPSHOT.Snapshot_Copy_Valid := FALSE;
    GVL_RUNTIME_SNAPSHOT.Snapshot_Isolation_Valid := FALSE;

    GVL_RUNTIME_SNAPSHOT.Snapshot_Runtime_Authority_Valid := FALSE;

    GVL_RUNTIME_SNAPSHOT.Snapshot_Last_Error_Code := L_Error_Code;
    GVL_RUNTIME_SNAPSHOT.Snapshot_Last_Error_Text := L_Error_Text;
END_IF;
END_PROGRAM

(* ---- PRG_Safety_Domain.st ---- *)
PROGRAM PRG_Safety_Domain
// SEMANTIC DOMAIN WRAPPER
// PRESERVES ORIGINAL EXECUTION ORDER
// NO EXECUTION SEMANTICS MUTATION

PRG_Safety();
PRG_Safety_Operator();
PRG_Safety_Shutdown();
PRG_Safety_Recovery();

PRG_Physical_SafeState_Lattice_Governor();
PRG_CrossDomain_FailSafe_Closure_Governor();

PRG_Safety_Observability_Truth_Governor();
PRG_Physical_Safety_Projection_Governor();

END_PROGRAM

(* ---- PRG_Safety_Operator.st ---- *)
PROGRAM PRG_Safety_Operator
VAR
    fbSafetyWorkflow : FB_Safety_Workflow_Manager;
END_VAR

// Operator / test / recover workflow ownership.

fbSafetyWorkflow(
    VI_System_Time_MS := GVL_TIME_SERVICE.G_Now_MS,
    VI_Water_Selective_Recover := GVL_INTENT_USER.I_Water_Selective_Recover,
    VI_Gas_Selective_Recover := GVL_INTENT_USER.I_Gas_Selective_Recover,
    VI_Water_Valve_Test_Open := GVL_INTENT_USER.I_Water_Valve_Test_Open,
    VI_Water_Valve_Test_Close := GVL_INTENT_USER.I_Water_Valve_Test_Close,
    VI_Water_Valve_Test_Confirm := GVL_INTENT_USER.I_Water_Valve_Test_Confirm,
    VI_Gas_Valve_Test_Open := GVL_INTENT_USER.I_Gas_Valve_Test_Open,
    VI_Gas_Valve_Test_Close := GVL_INTENT_USER.I_Gas_Valve_Test_Close,
    VI_Gas_Valve_Test_Confirm := GVL_INTENT_USER.I_Gas_Valve_Test_Confirm
);

// propagate test timeout safety actions
IF fbSafetyWorkflow.VO_Water_Test_Timeout_Close_Required THEN
    GVL_INTENT_SAFETY.I_Test_Timeout_Water_Close := TRUE;
END_IF;

IF fbSafetyWorkflow.VO_Gas_Test_Timeout_Close_Required THEN
    GVL_INTENT_SAFETY.I_Test_Timeout_Gas_Close := TRUE;
END_IF;

// move recovery manual confirm here
IF GVL_INTENT_USER.I_Reset_Errors THEN
    GVL_SAFETY_RECOVERY.G_Recovery_Manual_Confirm := TRUE;
END_IF;

// >>> BULK_SYNC_ANCHOR: PRG_Safety_Operator <<<
END_PROGRAM

(* ---- PRG_Sensor_Consensus_Governor.st ---- *)
PROGRAM PRG_Sensor_Consensus_Governor
VAR
    L_Now_MS : UDINT;
    L_Consensus_Valid : BOOL := TRUE;
    L_Error_Code : UDINT := 0;
    L_Error_Text : STRING(160) := '';
    L_Consensus_Age_MS : UDINT;
END_VAR

L_Now_MS := GVL_STATUS.G_System_Time_MS;
L_Consensus_Valid := TRUE;
L_Error_Code := 0;
L_Error_Text := '';

// Fail-safe defaults.
GVL_SENSOR_CONSENSUS.Sensor_Consensus_Valid := FALSE;
GVL_SENSOR_CONSENSUS.Sensor_Consensus_Quarantine_Active := TRUE;
GVL_SENSOR_CONSENSUS.Sensor_Consensus_Lease_Expired := TRUE;
GVL_SENSOR_CONSENSUS.Sensor_Consensus_Freshness_Valid := FALSE;

GVL_SENSOR_CONSENSUS.Physics_Invariants_Satisfied := FALSE;
GVL_SENSOR_CONSENSUS.Cross_Sensor_Correlation_Valid := FALSE;
GVL_SENSOR_CONSENSUS.Telemetry_Plausibility_Valid := FALSE;

IF GVL_SENSOR_CONSENSUS.Sensor_Replay_Suspected THEN
    L_Consensus_Valid := FALSE;
    L_Error_Code := 22000;
    L_Error_Text := 'Sensor replay suspected';
END_IF;

IF L_Consensus_Valid
AND GVL_SENSOR_CONSENSUS.Sensor_Partition_Detected THEN
    L_Consensus_Valid := FALSE;
    L_Error_Code := 22001;
    L_Error_Text := 'Sensor partition detected';
END_IF;

IF L_Consensus_Valid
AND GVL_SENSOR_CONSENSUS.Sensor_Hallucination_Suspected THEN
    L_Consensus_Valid := FALSE;
    L_Error_Code := 22002;
    L_Error_Text := 'Sensor hallucination suspected';
END_IF;

IF L_Consensus_Valid
AND GVL_SENSOR_CONSENSUS.Cross_Sensor_Divergence_Detected THEN
    L_Consensus_Valid := FALSE;
    L_Error_Code := 22003;
    L_Error_Text := 'Cross sensor divergence detected';
END_IF;

IF L_Consensus_Valid
AND GVL_SENSOR_CONSENSUS.Sensor_Drift_Detected THEN
    L_Consensus_Valid := FALSE;
    L_Error_Code := 22004;
    L_Error_Text := 'Sensor drift detected';
END_IF;

IF L_Consensus_Valid
AND GVL_SENSOR_CONSENSUS.Sensor_Oscillation_Detected THEN
    L_Consensus_Valid := FALSE;
    L_Error_Code := 22005;
    L_Error_Text := 'Sensor oscillation detected';
END_IF;

IF L_Consensus_Valid
AND GVL_SENSOR_CONSENSUS.Sensor_Stuck_State_Detected THEN
    L_Consensus_Valid := FALSE;
    L_Error_Code := 22006;
    L_Error_Text := 'Sensor stuck state detected';
END_IF;

// Physics invariants.
IF L_Consensus_Valid
AND NOT GVL_SENSOR_CONSENSUS.Flow_Response_Valid THEN
    L_Consensus_Valid := FALSE;
    L_Error_Code := 22010;
    L_Error_Text := 'Flow response invalid';
END_IF;

IF L_Consensus_Valid
AND NOT GVL_SENSOR_CONSENSUS.Pressure_Response_Valid THEN
    L_Consensus_Valid := FALSE;
    L_Error_Code := 22011;
    L_Error_Text := 'Pressure response invalid';
END_IF;

IF L_Consensus_Valid
AND NOT GVL_SENSOR_CONSENSUS.Airflow_Response_Valid THEN
    L_Consensus_Valid := FALSE;
    L_Error_Code := 22012;
    L_Error_Text := 'Airflow response invalid';
END_IF;

IF L_Consensus_Valid
AND NOT GVL_SENSOR_CONSENSUS.Current_Signature_Valid THEN
    L_Consensus_Valid := FALSE;
    L_Error_Code := 22013;
    L_Error_Text := 'Current signature invalid';
END_IF;

// Consensus freshness.
L_Consensus_Age_MS :=
    L_Now_MS - GVL_SENSOR_CONSENSUS.Last_Consensus_Update_MS;

IF L_Consensus_Valid
AND (L_Consensus_Age_MS > 5000) THEN
    L_Consensus_Valid := FALSE;
    L_Error_Code := 22020;
    L_Error_Text := 'Sensor consensus stale';
END_IF;

IF L_Consensus_Valid THEN
    GVL_SENSOR_CONSENSUS.Sensor_Consensus_Valid := TRUE;
    GVL_SENSOR_CONSENSUS.Sensor_Consensus_Quarantine_Active := FALSE;
    GVL_SENSOR_CONSENSUS.Sensor_Consensus_Lease_Expired := FALSE;
    GVL_SENSOR_CONSENSUS.Sensor_Consensus_Freshness_Valid := TRUE;

    GVL_SENSOR_CONSENSUS.Physics_Invariants_Satisfied := TRUE;
    GVL_SENSOR_CONSENSUS.Cross_Sensor_Correlation_Valid := TRUE;
    GVL_SENSOR_CONSENSUS.Telemetry_Plausibility_Valid := TRUE;

    GVL_SENSOR_CONSENSUS.Sensor_Consensus_Epoch :=
        GVL_SENSOR_CONSENSUS.Sensor_Consensus_Epoch + 1;

    GVL_SENSOR_CONSENSUS.Last_Consensus_Update_MS := L_Now_MS;

    GVL_SENSOR_CONSENSUS.Sensor_Consensus_Last_Error_Code := 0;
    GVL_SENSOR_CONSENSUS.Sensor_Consensus_Last_Error_Text := '';
ELSE
    GVL_SENSOR_CONSENSUS.Sensor_Consensus_Valid := FALSE;
    GVL_SENSOR_CONSENSUS.Sensor_Consensus_Quarantine_Active := TRUE;
    GVL_SENSOR_CONSENSUS.Sensor_Consensus_Lease_Expired := TRUE;
    GVL_SENSOR_CONSENSUS.Sensor_Consensus_Freshness_Valid := FALSE;

    GVL_SENSOR_CONSENSUS.Sensor_Consensus_Last_Error_Code := L_Error_Code;
    GVL_SENSOR_CONSENSUS.Sensor_Consensus_Last_Error_Text := L_Error_Text;

    GVL_SENSOR_CONSENSUS.Sensor_Consensus_Invalidation_Count :=
        GVL_SENSOR_CONSENSUS.Sensor_Consensus_Invalidation_Count + 1;
END_IF;

END_PROGRAM

(* ---- PRG_System_Diagnostics_Ext.st ---- *)
PROGRAM PRG_System_Diagnostics_Ext
VAR
    L_Error_Heating : BOOL;
    L_Error_Safety : BOOL;
    L_Error_IO : BOOL;

    L_Delta_Time : REAL;
    L_Now : UDINT;
    L_Last : UDINT;

    // cycle stats
    L_Cycle_MS : UDINT;
    L_Prev_Overrun : BOOL;
    L_Prev_Critical : BOOL;
    fbLog : FB_LogEvent;
END_VAR

L_Now := GVL_TIME_SERVICE.G_Now_MS;
L_Last := GVL_DIAGNOSTICS_EXT.G_Last_Update_Time;

// ===============================
// CYCLE INTERVAL MEASUREMENT
// ===============================
IF L_Last = 0 THEN
    L_Cycle_MS := GVL_DIAGNOSTICS_EXT.G_Cycle_Expected_MS;
ELSE
    IF L_Now >= L_Last THEN
        L_Cycle_MS := L_Now - L_Last;
    ELSE
        L_Cycle_MS := (4294967295 - L_Last) + L_Now + 1;
    END_IF;
END_IF;

GVL_DIAGNOSTICS_EXT.G_Last_Update_Time := L_Now;
GVL_DIAGNOSTICS_EXT.G_Cycle_Last_MS := L_Cycle_MS;

// min/max
IF (GVL_DIAGNOSTICS_EXT.G_Cycle_Min_MS = 0) OR (L_Cycle_MS < GVL_DIAGNOSTICS_EXT.G_Cycle_Min_MS) THEN
    GVL_DIAGNOSTICS_EXT.G_Cycle_Min_MS := L_Cycle_MS;
END_IF;

IF L_Cycle_MS > GVL_DIAGNOSTICS_EXT.G_Cycle_Max_MS THEN
    GVL_DIAGNOSTICS_EXT.G_Cycle_Max_MS := L_Cycle_MS;
END_IF;

// average (incremental)
GVL_DIAGNOSTICS_EXT.G_Cycle_Sample_Count := GVL_DIAGNOSTICS_EXT.G_Cycle_Sample_Count + 1;
GVL_DIAGNOSTICS_EXT.G_Cycle_Avg_MS :=
    GVL_DIAGNOSTICS_EXT.G_Cycle_Avg_MS +
    (UDINT_TO_REAL(L_Cycle_MS) - GVL_DIAGNOSTICS_EXT.G_Cycle_Avg_MS) /
    UDINT_TO_REAL(GVL_DIAGNOSTICS_EXT.G_Cycle_Sample_Count);

// ===============================
// OVERRUN / CRITICAL DETECTION
// ===============================
GVL_DIAGNOSTICS_EXT.G_Cycle_Overrun_Active := (L_Cycle_MS > GVL_DIAGNOSTICS_EXT.G_Cycle_Warning_MS);
GVL_DIAGNOSTICS_EXT.G_Cycle_Critical_Active := (L_Cycle_MS > GVL_DIAGNOSTICS_EXT.G_Cycle_Critical_MS);

IF GVL_DIAGNOSTICS_EXT.G_Cycle_Overrun_Active THEN
    GVL_DIAGNOSTICS_EXT.G_Cycle_Overrun_Count := GVL_DIAGNOSTICS_EXT.G_Cycle_Overrun_Count + 1;
    GVL_DIAGNOSTICS_EXT.G_Cycle_Last_Overrun_MS := L_Cycle_MS;
    GVL_DIAGNOSTICS_EXT.G_Cycle_Last_Overrun_Time_MS := L_Now;
END_IF;

IF GVL_DIAGNOSTICS_EXT.G_Cycle_Critical_Active THEN
    GVL_DIAGNOSTICS_EXT.G_Cycle_Critical_Count := GVL_DIAGNOSTICS_EXT.G_Cycle_Critical_Count + 1;
END_IF;

// edge logging
IF GVL_DIAGNOSTICS_EXT.G_Cycle_Overrun_Active AND NOT L_Prev_Overrun THEN
    fbLog(
        VI_Event_Type := 2001,
        VI_Timestamp := L_Now,
        VI_Param1 := L_Cycle_MS,
        VI_Param2 := GVL_DIAGNOSTICS_EXT.G_Cycle_Overrun_Count
    );
END_IF;

IF GVL_DIAGNOSTICS_EXT.G_Cycle_Critical_Active AND NOT L_Prev_Critical THEN
    fbLog(
        VI_Event_Type := 2002,
        VI_Timestamp := L_Now,
        VI_Param1 := L_Cycle_MS,
        VI_Param2 := GVL_DIAGNOSTICS_EXT.G_Cycle_Critical_Count
    );
END_IF;

L_Prev_Overrun := GVL_DIAGNOSTICS_EXT.G_Cycle_Overrun_Active;
L_Prev_Critical := GVL_DIAGNOSTICS_EXT.G_Cycle_Critical_Active;

// ===============================
// EXISTING HEALTH LOGIC
// ===============================
IF L_Last = 0 THEN
    L_Delta_Time := 0.1;
ELSE
    L_Delta_Time := UDINT_TO_REAL(L_Cycle_MS) / 1000.0;
END_IF;

L_Error_Heating := GVL_STATE.G_Heating_Subsystem_Degraded;

// Extended diagnostics must use authoritative safety truth and latches,
// not stale projected GVL_STATE.G_Safety_*_Alarm compatibility fields.
L_Error_Safety :=
    GVL_HEALTH_BRIDGE.G_Gas_Detected OR
    GVL_HEALTH_BRIDGE.G_CO_Alarm_Level OR
    GVL_HEALTH_BRIDGE.G_Leak_Detected OR
    GVL_HEALTH_BRIDGE.G_Smoke_Detected OR
    GVL_STATE.G_Safety_Gas_Latched OR
    GVL_STATE.G_Safety_Leak_Latched OR
    GVL_STATE.G_Safety_Smoke_Latched;

L_Error_IO := GVL_STATE.G_Heating_IO_Fault;

IF L_Error_Heating THEN
    GVL_DIAGNOSTICS_EXT.G_Error_Count_Heating := GVL_DIAGNOSTICS_EXT.G_Error_Count_Heating + 1;
    GVL_DIAGNOSTICS_EXT.G_Last_Error_Time_Heating := L_Now;
    GVL_DIAGNOSTICS_EXT.G_Health_Heating := GVL_DIAGNOSTICS_EXT.G_Health_Heating - (0.5 * L_Delta_Time);
ELSE
    GVL_DIAGNOSTICS_EXT.G_Health_Heating := GVL_DIAGNOSTICS_EXT.G_Health_Heating + (0.1 * L_Delta_Time);
END_IF;

IF L_Error_Safety THEN
    GVL_DIAGNOSTICS_EXT.G_Error_Count_Safety := GVL_DIAGNOSTICS_EXT.G_Error_Count_Safety + 1;
    GVL_DIAGNOSTICS_EXT.G_Last_Error_Time_Safety := L_Now;
    GVL_DIAGNOSTICS_EXT.G_Health_Safety := GVL_DIAGNOSTICS_EXT.G_Health_Safety - (1.0 * L_Delta_Time);
ELSE
    GVL_DIAGNOSTICS_EXT.G_Health_Safety := GVL_DIAGNOSTICS_EXT.G_Health_Safety + (0.2 * L_Delta_Time);
END_IF;

IF L_Error_IO THEN
    GVL_DIAGNOSTICS_EXT.G_Error_Count_IO := GVL_DIAGNOSTICS_EXT.G_Error_Count_IO + 1;
    GVL_DIAGNOSTICS_EXT.G_Last_Error_Time_IO := L_Now;
    GVL_DIAGNOSTICS_EXT.G_Health_IO := GVL_DIAGNOSTICS_EXT.G_Health_IO - (0.5 * L_Delta_Time);
ELSE
    GVL_DIAGNOSTICS_EXT.G_Health_IO := GVL_DIAGNOSTICS_EXT.G_Health_IO + (0.1 * L_Delta_Time);
END_IF;

// clamp
IF GVL_DIAGNOSTICS_EXT.G_Health_Heating < 0.0 THEN GVL_DIAGNOSTICS_EXT.G_Health_Heating := 0.0; END_IF;
IF GVL_DIAGNOSTICS_EXT.G_Health_Heating > 1.0 THEN GVL_DIAGNOSTICS_EXT.G_Health_Heating := 1.0; END_IF;

IF GVL_DIAGNOSTICS_EXT.G_Health_Safety < 0.0 THEN GVL_DIAGNOSTICS_EXT.G_Health_Safety := 0.0; END_IF;
IF GVL_DIAGNOSTICS_EXT.G_Health_Safety > 1.0 THEN GVL_DIAGNOSTICS_EXT.G_Health_Safety := 1.0; END_IF;

IF GVL_DIAGNOSTICS_EXT.G_Health_IO < 0.0 THEN GVL_DIAGNOSTICS_EXT.G_Health_IO := 0.0; END_IF;
IF GVL_DIAGNOSTICS_EXT.G_Health_IO > 1.0 THEN GVL_DIAGNOSTICS_EXT.G_Health_IO := 1.0; END_IF;

END_PROGRAM

(* ---- PRG_System_History.st ---- *)
PROGRAM PRG_System_History
VAR
    fbHistoryManager : FB_History_Manager;
    L_History_Event : ST_History_Record;
    L_History_Write_Event : BOOL;
    L_Last_System_Mode : E_System_Operating_Mode;
    L_Last_Root_Cause : E_System_Root_Cause;
    L_Last_First_Fault_Source : INT;
    L_Last_Operator_Journal_Seq : UDINT;
    L_Last_Event_Code : UDINT;
    L_Last_Event_Value : REAL;
    L_Last_Event_Time_MS : UDINT;
END_VAR

L_History_Write_Event := FALSE;
L_History_Event.timestamp_ms := GVL_TIME_SERVICE.G_Now_MS;
L_History_Event.event_code := 0;
L_History_Event.event_value := 0.0;
L_History_Event.unit := 0;
L_History_Event.zone_id := 0;
L_History_Event.operator_id := 'SYSTEM';
L_History_Event.priority := E_ALERT_PRIORITY.ALERT_PRIORITY_HIGH;

IF GVL_STATE.G_System_Mode <> L_Last_System_Mode THEN
    L_History_Write_Event := TRUE;
    L_History_Event.event_code := 1101;
    L_History_Event.event_value := TO_REAL(TO_INT(GVL_STATE.G_System_Mode));
    L_History_Event.unit := 1;
    L_History_Event.zone_id := 0;
    L_History_Event.priority := E_ALERT_PRIORITY.ALERT_PRIORITY_HIGH;
    L_Last_System_Mode := GVL_STATE.G_System_Mode;

ELSIF GVL_SYSTEM_HEALTH.G_Root_Cause <> L_Last_Root_Cause THEN
    L_History_Write_Event := TRUE;
    L_History_Event.event_code := 1102;
    L_History_Event.event_value := TO_REAL(TO_INT(GVL_SYSTEM_HEALTH.G_Root_Cause));
    L_History_Event.unit := 2;
    L_History_Event.zone_id := TO_BYTE(GVL_SYSTEM_HEALTH.G_First_Fault_Source);
    L_History_Event.priority := E_ALERT_PRIORITY.ALERT_PRIORITY_HIGH;
    L_Last_Root_Cause := GVL_SYSTEM_HEALTH.G_Root_Cause;

ELSIF GVL_SYSTEM_HEALTH.G_First_Fault_Source <> L_Last_First_Fault_Source THEN
    L_History_Write_Event := TRUE;
    L_History_Event.event_code := 1103;
    L_History_Event.event_value := TO_REAL(GVL_SYSTEM_HEALTH.G_First_Fault_Source);
    L_History_Event.unit := 3;
    L_History_Event.zone_id := TO_BYTE(GVL_SYSTEM_HEALTH.G_First_Fault_Source);
    L_History_Event.priority := E_ALERT_PRIORITY.ALERT_PRIORITY_HIGH;
    L_Last_First_Fault_Source := GVL_SYSTEM_HEALTH.G_First_Fault_Source;

ELSIF GVL_STATUS.G_Current_Scenario <> GVL_STATUS.G_Previous_Scenario THEN
    L_History_Write_Event := TRUE;
    L_History_Event.event_code := 1001;
    L_History_Event.event_value := TO_REAL(GVL_STATUS.G_Current_Scenario);
    L_History_Event.unit := 4;
    L_History_Event.zone_id := 0;
    L_History_Event.priority := E_ALERT_PRIORITY.ALERT_PRIORITY_HIGH;
    GVL_STATUS.G_Previous_Scenario := GVL_STATUS.G_Current_Scenario;

ELSIF GVL_STATUS.G_Diagnostics.Alarm_Event_Pulse THEN
    L_History_Write_Event := TRUE;
    L_History_Event.event_code := TO_WORD(GVL_STATUS.G_Diagnostics.Alarm_Event_Code);
    L_History_Event.event_value := GVL_STATUS.G_Diagnostics.Alarm_Event_Value;
    L_History_Event.unit := 10;
    L_History_Event.zone_id := 0;
    L_History_Event.priority := E_ALERT_PRIORITY.ALERT_PRIORITY_HIGH;

ELSIF GVL_STATUS.G_Diagnostics.Operator_Journal_Event_Seq <> L_Last_Operator_Journal_Seq THEN
    L_History_Write_Event := TRUE;
    L_History_Event.event_code := 1301;
    L_History_Event.event_value := TO_REAL(GVL_STATUS.G_Diagnostics.Operator_Journal_Event_Seq);
    L_History_Event.unit := 20;
    L_History_Event.zone_id := 0;
    L_History_Event.priority := E_ALERT_PRIORITY.ALERT_PRIORITY_HIGH;
    L_Last_Operator_Journal_Seq := GVL_STATUS.G_Diagnostics.Operator_Journal_Event_Seq;
END_IF;

IF L_History_Write_Event THEN
    IF (L_History_Event.event_code = L_Last_Event_Code)
       AND (ABS(L_History_Event.event_value - L_Last_Event_Value) < 0.001)
       AND (GVL_TIME_SERVICE.G_Now_MS - L_Last_Event_Time_MS < 5000) THEN
        L_History_Write_Event := FALSE;
    ELSE
        L_Last_Event_Code := L_History_Event.event_code;
        L_Last_Event_Value := L_History_Event.event_value;
        L_Last_Event_Time_MS := GVL_TIME_SERVICE.G_Now_MS;
    END_IF;
END_IF;

fbHistoryManager(
    VI_System_Time_MS := GVL_TIME_SERVICE.G_Now_MS,
    VI_Write_Event := L_History_Write_Event,
    VI_Event := L_History_Event
);

END_PROGRAM

(* ---- PRG_System_Intent.st ---- *)
PROGRAM PRG_System_Intent
VAR
    fbSystemIntentPublisher : FB_System_Intent_Publisher;
    L_Gateway_Writes_Allowed : BOOL;
END_VAR

// Extracted from PRG_System (Phase 5A).
// Idempotent projection: safe to run while legacy call still exists.
L_Gateway_Writes_Allowed :=
    NOT GVL_STATUS.G_Diagnostics.Dangerous_Action_Pending_Confirm AND
    NOT GVL_STATUS.G_Diagnostics.Operator_Action_Blocked AND
    NOT GVL_STATUS.G_Diagnostics.User_Access_Denied;

fbSystemIntentPublisher(
    VI_System_Time_MS := GVL_TIME_SERVICE.G_Now_MS,
    VI_Gateway_Writes_Allowed := L_Gateway_Writes_Allowed
);

END_PROGRAM

(* ---- PRG_Telemetry_Causality_Governor.st ---- *)
PROGRAM PRG_Telemetry_Causality_Governor
VAR
    L_Now_MS : UDINT;
    L_Causality_Valid : BOOL := TRUE;
    L_Error_Code : UDINT := 0;
    L_Error_Text : STRING(160) := '';
    L_Ack_Age_MS : UDINT;
    L_Convergence_Age_MS : UDINT;
    L_Stable_Dwell_MS : UDINT;
    L_Consensus_Age_MS : UDINT;
END_VAR

L_Now_MS := GVL_STATUS.G_System_Time_MS;
L_Causality_Valid := TRUE;
L_Error_Code := 0;
L_Error_Text := '';

GVL_TELEMETRY.Telemetry_Runtime_Valid := FALSE;
GVL_TELEMETRY.Telemetry_Freshness_Valid := FALSE;
GVL_TELEMETRY.Command_Telemetry_Causality_Valid := FALSE;
GVL_TELEMETRY.Actuator_Feedback_Valid := FALSE;
GVL_TELEMETRY.Actuator_Feedback_Fresh := FALSE;
GVL_TELEMETRY.Physical_Effect_Confirmed := FALSE;
GVL_TELEMETRY.Physical_Effect_Finalized := FALSE;
GVL_TELEMETRY.Physical_Target_Converged := FALSE;
GVL_TELEMETRY.Physical_Stable_Window_OK := FALSE;
GVL_TELEMETRY.Command_Telemetry_Divergence_Detected := TRUE;

GVL_TELEMETRY.Command_Epoch := ULINT_TO_UDINT(GVL_OUTPUT_EPOCH.Output_Publication_Epoch);

IF NOT GVL_OUTPUT_EPOCH.Output_Publication_Valid THEN
    L_Causality_Valid := FALSE;
    L_Error_Code := 21000;
    L_Error_Text := 'Telemetry causality output publication invalid';
END_IF;

IF L_Causality_Valid AND NOT GVL_OUTPUT_EPOCH.Output_Runtime_Epoch_Valid THEN
    L_Causality_Valid := FALSE;
    L_Error_Code := 21001;
    L_Error_Text := 'Telemetry causality runtime epoch invalid';
END_IF;

IF L_Causality_Valid AND GVL_OUTPUT_EPOCH.Output_Lease_Expired THEN
    L_Causality_Valid := FALSE;
    L_Error_Code := 21002;
    L_Error_Text := 'Telemetry causality output lease expired';
END_IF;

IF L_Causality_Valid AND GVL_OUTPUT_EPOCH.Output_Forced_Safe_Decay THEN
    L_Causality_Valid := FALSE;
    L_Error_Code := 21003;
    L_Error_Text := 'Telemetry causality output forced safe decay';
END_IF;

IF L_Causality_Valid AND (GVL_TELEMETRY.Telemetry_Epoch <> GVL_TELEMETRY.Command_Epoch) THEN
    L_Causality_Valid := FALSE;
    L_Error_Code := 21010;
    L_Error_Text := 'Telemetry epoch does not match command epoch';
END_IF;

IF L_Causality_Valid AND (GVL_TELEMETRY.Telemetry_Epoch < GVL_TELEMETRY.Last_Acknowledged_Command_Epoch) THEN
    GVL_TELEMETRY.Telemetry_Replay_Suspected := TRUE;

    L_Causality_Valid := FALSE;
    L_Error_Code := 21011;
    L_Error_Text := 'Telemetry epoch replay suspected';
END_IF;

L_Ack_Age_MS := L_Now_MS - GVL_TELEMETRY.Last_Physical_Ack_Time_MS;

IF L_Causality_Valid AND (L_Ack_Age_MS > 5000) THEN
    L_Causality_Valid := FALSE;
    L_Error_Code := 21020;
    L_Error_Text := 'Physical acknowledgement stale';
END_IF;

L_Convergence_Age_MS := L_Now_MS - GVL_TELEMETRY.Last_Physical_Convergence_MS;

IF L_Causality_Valid AND (L_Convergence_Age_MS > 10000) THEN
    L_Causality_Valid := FALSE;
    L_Error_Code := 21021;
    L_Error_Text := 'Physical convergence stale';
END_IF;

L_Stable_Dwell_MS :=
    L_Now_MS - GVL_TELEMETRY.Last_Physical_Convergence_MS;

IF L_Causality_Valid AND (L_Stable_Dwell_MS < 3000) THEN
    L_Causality_Valid := FALSE;
    L_Error_Code := 21030;
    L_Error_Text := 'Physical stabilization dwell window incomplete';
END_IF;

IF L_Causality_Valid
AND GVL_TELEMETRY.Physical_Oscillation_Detected THEN
    L_Causality_Valid := FALSE;
    L_Error_Code := 21031;
    L_Error_Text := 'Physical oscillation detected';
END_IF;

IF L_Causality_Valid
AND GVL_TELEMETRY.Physical_Transition_Active THEN
    L_Causality_Valid := FALSE;
    L_Error_Code := 21032;
    L_Error_Text := 'Physical transition still active';
END_IF;

IF L_Causality_Valid
AND GVL_TELEMETRY.Physical_Convergence_Replay_Suspected THEN
    L_Causality_Valid := FALSE;
    L_Error_Code := 21033;
    L_Error_Text := 'Physical convergence replay suspected';
END_IF;

L_Consensus_Age_MS :=
    L_Now_MS - GVL_SENSOR_CONSENSUS.Last_Consensus_Update_MS;

IF L_Causality_Valid
AND (L_Consensus_Age_MS > 5000) THEN
    L_Causality_Valid := FALSE;
    L_Error_Code := 21040;
    L_Error_Text := 'Sensor consensus stale';
END_IF;

IF L_Causality_Valid
AND NOT GVL_SENSOR_CONSENSUS.Sensor_Consensus_Valid THEN
    L_Causality_Valid := FALSE;
    L_Error_Code := 21041;
    L_Error_Text := 'Sensor consensus invalid';
END_IF;

IF L_Causality_Valid
AND NOT GVL_SENSOR_CONSENSUS.Physics_Invariants_Satisfied THEN
    L_Causality_Valid := FALSE;
    L_Error_Code := 21042;
    L_Error_Text := 'Physics invariants violated';
END_IF;

IF L_Causality_Valid
AND NOT GVL_SENSOR_CONSENSUS.Cross_Sensor_Correlation_Valid THEN
    L_Causality_Valid := FALSE;
    L_Error_Code := 21043;
    L_Error_Text := 'Cross sensor correlation invalid';
END_IF;

IF L_Causality_Valid
AND NOT GVL_SENSOR_CONSENSUS.Telemetry_Plausibility_Valid THEN
    L_Causality_Valid := FALSE;
    L_Error_Code := 21044;
    L_Error_Text := 'Telemetry plausibility invalid';
END_IF;

IF L_Causality_Valid
AND (GVL_SENSOR_CONSENSUS.Sensor_Drift_Detected
     OR GVL_SENSOR_CONSENSUS.Sensor_Partition_Detected
     OR GVL_SENSOR_CONSENSUS.Sensor_Hallucination_Suspected
     OR GVL_SENSOR_CONSENSUS.Cross_Sensor_Divergence_Detected
     OR GVL_SENSOR_CONSENSUS.Sensor_Oscillation_Detected
     OR GVL_SENSOR_CONSENSUS.Sensor_Stuck_State_Detected
     OR GVL_SENSOR_CONSENSUS.Sensor_Replay_Suspected) THEN

    L_Causality_Valid := FALSE;
    L_Error_Code := 21045;
    L_Error_Text := 'Sensor consensus divergence detected';
END_IF;

IF L_Causality_Valid THEN
    GVL_TELEMETRY.Telemetry_Runtime_Valid := TRUE;
    GVL_TELEMETRY.Telemetry_Freshness_Valid := TRUE;
    GVL_TELEMETRY.Telemetry_Lease_Expired := FALSE;
    GVL_TELEMETRY.Telemetry_Quarantine_Active := FALSE;

    GVL_TELEMETRY.Command_Telemetry_Causality_Valid := TRUE;
    GVL_TELEMETRY.Command_Telemetry_Divergence_Detected := FALSE;

    GVL_TELEMETRY.Actuator_Feedback_Valid := TRUE;
    GVL_TELEMETRY.Actuator_Feedback_Fresh := TRUE;
    GVL_TELEMETRY.Physical_Effect_Confirmed := TRUE;

    GVL_TELEMETRY.Physical_Target_Converged := TRUE;
    GVL_TELEMETRY.Physical_Stable_Window_OK := TRUE;
    GVL_TELEMETRY.Physical_Effect_Finalized := TRUE;

    GVL_TELEMETRY.Last_Acknowledged_Command_Epoch := GVL_TELEMETRY.Command_Epoch;

    GVL_TELEMETRY.Telemetry_Last_Error_Code := 0;
    GVL_TELEMETRY.Telemetry_Last_Error_Text := '';
ELSE
    GVL_TELEMETRY.Telemetry_Runtime_Valid := FALSE;
    GVL_TELEMETRY.Telemetry_Freshness_Valid := FALSE;
    GVL_TELEMETRY.Telemetry_Lease_Expired := TRUE;
    GVL_TELEMETRY.Telemetry_Quarantine_Active := TRUE;

    GVL_TELEMETRY.Command_Telemetry_Causality_Valid := FALSE;
    GVL_TELEMETRY.Command_Telemetry_Divergence_Detected := TRUE;

    GVL_TELEMETRY.Telemetry_Last_Error_Code := L_Error_Code;
    GVL_TELEMETRY.Telemetry_Last_Error_Text := L_Error_Text;
    GVL_TELEMETRY.Telemetry_Invalidation_Count :=
        GVL_TELEMETRY.Telemetry_Invalidation_Count + 1;
END_IF;

END_PROGRAM
